# B&R Automation Studio project CControl_Gschneitner (part 4)

#### fbTrockVariante.st - Auswertung der Anlagenkonfiguration mit Ausgabe einer Nummer und eines Textes
```iecst
(********************************************************************
 * COPYRIGHT -- LASCO Heu- und Forsttechnik GmbH
 ********************************************************************
 * Library: LascoTrock
 * Datei: fbTrockVariante.st
 * Autor: Rudolf Lachner
 * Erstellt: 12. Februar 2015
 ********************************************************************
 * Implementierung der Library LascoTrock
 ********************************************************************)

(* Auswertung der Anlagenkonfiguration mit Ausgabe einer Nummer und eines Textes *)
FUNCTION_BLOCK fbTrockVariante

	IF Freigabe THEN

		IF (Ventilator1 AND NOT Ventilator2 AND NOT Luftentfeuchter AND NOT Warmluftofen AND NOT BetriebsmldgWarmluftofen AND NOT BetriebsmldgScheitholzofen AND NOT Brandschutzklappe AND NOT Umschaltklappe) THEN
			VarianteNr 	:= 1;
		ELSIF (Ventilator1 AND NOT Ventilator2 AND NOT Luftentfeuchter AND NOT Warmluftofen AND NOT BetriebsmldgWarmluftofen AND NOT BetriebsmldgScheitholzofen AND NOT Brandschutzklappe AND Umschaltklappe) THEN
			VarianteNr 	:= 2;
		ELSIF (Ventilator1 AND NOT Ventilator2 AND NOT Luftentfeuchter AND NOT Warmluftofen AND NOT BetriebsmldgWarmluftofen AND BetriebsmldgScheitholzofen AND NOT Brandschutzklappe AND NOT Umschaltklappe) THEN
			VarianteNr 	:= 3;
		ELSIF (Ventilator1 AND NOT Ventilator2 AND NOT Luftentfeuchter AND NOT Warmluftofen AND NOT BetriebsmldgWarmluftofen AND BetriebsmldgScheitholzofen AND NOT Brandschutzklappe AND Umschaltklappe) THEN
			VarianteNr 	:= 4;
		ELSIF (Ventilator1 AND NOT Ventilator2 AND NOT Luftentfeuchter AND NOT Warmluftofen AND NOT BetriebsmldgWarmluftofen AND BetriebsmldgScheitholzofen AND Brandschutzklappe AND NOT Umschaltklappe) THEN
			VarianteNr 	:= 5;
		ELSIF (Ventilator1 AND NOT Ventilator2 AND NOT Luftentfeuchter AND NOT Warmluftofen AND NOT BetriebsmldgWarmluftofen AND BetriebsmldgScheitholzofen AND Brandschutzklappe AND Umschaltklappe) THEN
			VarianteNr 	:= 6;
		ELSIF (Ventilator1 AND NOT Ventilator2 AND NOT Luftentfeuchter AND NOT Warmluftofen AND BetriebsmldgWarmluftofen AND NOT BetriebsmldgScheitholzofen AND NOT Brandschutzklappe AND NOT Umschaltklappe) THEN
			VarianteNr 	:= 7;
		ELSIF (Ventilator1 AND NOT Ventilator2 AND NOT Luftentfeuchter AND NOT Warmluftofen AND BetriebsmldgWarmluftofen AND NOT BetriebsmldgScheitholzofen AND NOT Brandschutzklappe AND Umschaltklappe) THEN
			VarianteNr 	:= 8;
		ELSIF (Ventilator1 AND NOT Ventilator2 AND NOT Luftentfeuchter AND NOT Warmluftofen AND BetriebsmldgWarmluftofen AND NOT BetriebsmldgScheitholzofen AND Brandschutzklappe AND NOT Umschaltklappe) THEN
			VarianteNr 	:= 9;
		ELSIF (Ventilator1 AND NOT Ventilator2 AND NOT Luftentfeuchter AND NOT Warmluftofen AND BetriebsmldgWarmluftofen AND NOT BetriebsmldgScheitholzofen AND Brandschutzklappe AND Umschaltklappe) THEN
			VarianteNr 	:= 10;
		ELSIF (Ventilator1 AND NOT Ventilator2 AND NOT Luftentfeuchter AND NOT Warmluftofen AND BetriebsmldgWarmluftofen AND BetriebsmldgScheitholzofen AND NOT Brandschutzklappe AND NOT Umschaltklappe) THEN
			VarianteNr 	:= 11;
		ELSIF (Ventilator1 AND NOT Ventilator2 AND NOT Luftentfeuchter AND NOT Warmluftofen AND BetriebsmldgWarmluftofen AND BetriebsmldgScheitholzofen AND NOT Brandschutzklappe AND Umschaltklappe) THEN
			VarianteNr 	:= 12;
		ELSIF (Ventilator1 AND NOT Ventilator2 AND NOT Luftentfeuchter AND NOT Warmluftofen AND BetriebsmldgWarmluftofen AND BetriebsmldgScheitholzofen AND Brandschutzklappe AND NOT Umschaltklappe) THEN
			VarianteNr 	:= 13;
		ELSIF (Ventilator1 AND NOT Ventilator2 AND NOT Luftentfeuchter AND NOT Warmluftofen AND BetriebsmldgWarmluftofen AND BetriebsmldgScheitholzofen AND Brandschutzklappe AND Umschaltklappe) THEN
			VarianteNr 	:= 14;
		ELSIF (Ventilator1 AND NOT Ventilator2 AND NOT Luftentfeuchter AND Warmluftofen AND NOT BetriebsmldgWarmluftofen AND NOT BetriebsmldgScheitholzofen AND NOT Brandschutzklappe AND NOT Umschaltklappe) THEN
			VarianteNr 	:= 15;
		ELSIF (Ventilator1 AND NOT Ventilator2 AND NOT Luftentfeuchter AND Warmluftofen AND NOT BetriebsmldgWarmluftofen AND NOT BetriebsmldgScheitholzofen AND NOT Brandschutzklappe AND Umschaltklappe) THEN
			VarianteNr 	:= 16;
		ELSIF (Ventilator1 AND NOT Ventilator2 AND NOT Luftentfeuchter AND Warmluftofen AND NOT BetriebsmldgWarmluftofen AND NOT BetriebsmldgScheitholzofen AND Brandschutzklappe AND NOT Umschaltklappe) THEN
			VarianteNr 	:= 17;
		ELSIF (Ventilator1 AND NOT Ventilator2 AND NOT Luftentfeuchter AND Warmluftofen AND NOT BetriebsmldgWarmluftofen AND NOT BetriebsmldgScheitholzofen AND Brandschutzklappe AND Umschaltklappe) THEN
			VarianteNr 	:= 18;
		ELSIF (Ventilator1 AND NOT Ventilator2 AND NOT Luftentfeuchter AND Warmluftofen AND NOT BetriebsmldgWarmluftofen AND BetriebsmldgScheitholzofen AND NOT Brandschutzklappe AND NOT Umschaltklappe) THEN
			VarianteNr 	:= 19;
		ELSIF (Ventilator1 AND NOT Ventilator2 AND NOT Luftentfeuchter AND Warmluftofen AND NOT BetriebsmldgWarmluftofen AND BetriebsmldgScheitholzofen AND NOT Brandschutzklappe AND Umschaltklappe) THEN
			VarianteNr 	:= 20;
		ELSIF (Ventilator1 AND NOT Ventilator2 AND NOT Luftentfeuchter AND Warmluftofen AND NOT BetriebsmldgWarmluftofen AND BetriebsmldgScheitholzofen AND Brandschutzklappe AND NOT Umschaltklappe) THEN
			VarianteNr 	:= 21;
		ELSIF (Ventilator1 AND NOT Ventilator2 AND NOT Luftentfeuchter AND Warmluftofen AND NOT BetriebsmldgWarmluftofen AND BetriebsmldgScheitholzofen AND Brandschutzklappe AND Umschaltklappe) THEN
			VarianteNr 	:= 22;
		ELSIF (Ventilator1 AND NOT Ventilator2 AND NOT Luftentfeuchter AND Warmluftofen AND BetriebsmldgWarmluftofen AND NOT BetriebsmldgScheitholzofen AND NOT Brandschutzklappe AND NOT Umschaltklappe) THEN
			VarianteNr 	:= 23;
		ELSIF (Ventilator1 AND NOT Ventilator2 AND NOT Luftentfeuchter AND Warmluftofen AND BetriebsmldgWarmluftofen AND NOT BetriebsmldgScheitholzofen AND NOT Brandschutzklappe AND Umschaltklappe) THEN
			VarianteNr 	:= 24;
		ELSIF (Ventilator1 AND NOT Ventilator2 AND NOT Luftentfeuchter AND Warmluftofen AND BetriebsmldgWarmluftofen AND NOT BetriebsmldgScheitholzofen AND Brandschutzklappe AND NOT Umschaltklappe) THEN
			VarianteNr 	:= 25;
		ELSIF (Ventilator1 AND NOT Ventilator2 AND NOT Luftentfeuchter AND Warmluftofen AND BetriebsmldgWarmluftofen AND NOT BetriebsmldgScheitholzofen AND Brandschutzklappe AND Umschaltklappe) THEN
			VarianteNr 	:= 26;
		ELSIF (Ventilator1 AND NOT Ventilator2 AND NOT Luftentfeuchter AND Warmluftofen AND BetriebsmldgWarmluftofen AND BetriebsmldgScheitholzofen AND NOT Brandschutzklappe AND NOT Umschaltklappe) THEN
			VarianteNr 	:= 27;
		ELSIF (Ventilator1 AND NOT Ventilator2 AND NOT Luftentfeuchter AND Warmluftofen AND BetriebsmldgWarmluftofen AND BetriebsmldgScheitholzofen AND NOT Brandschutzklappe AND Umschaltklappe) THEN
			VarianteNr 	:= 28;
		ELSIF (Ventilator1 AND NOT Ventilator2 AND NOT Luftentfeuchter AND Warmluftofen AND BetriebsmldgWarmluftofen AND BetriebsmldgScheitholzofen AND Brandschutzklappe AND NOT Umschaltklappe) THEN
			VarianteNr 	:= 29;
		ELSIF (Ventilator1 AND NOT Ventilator2 AND NOT Luftentfeuchter AND Warmluftofen AND BetriebsmldgWarmluftofen AND BetriebsmldgScheitholzofen AND Brandschutzklappe AND Umschaltklappe) THEN
			VarianteNr 	:= 30;
		ELSIF (Ventilator1 AND NOT Ventilator2 AND Luftentfeuchter AND NOT Warmluftofen AND NOT BetriebsmldgWarmluftofen AND NOT BetriebsmldgScheitholzofen AND NOT Brandschutzklappe AND NOT Umschaltklappe) THEN
			VarianteNr 	:= 31;
		ELSIF (Ventilator1 AND NOT Ventilator2 AND Luftentfeuchter AND NOT Warmluftofen AND NOT BetriebsmldgWarmluftofen AND NOT BetriebsmldgScheitholzofen AND NOT Brandschutzklappe AND Umschaltklappe) THEN
			VarianteNr 	:= 32;
		ELSIF (Ventilator1 AND NOT Ventilator2 AND Luftentfeuchter AND NOT Warmluftofen AND NOT BetriebsmldgWarmluftofen AND BetriebsmldgScheitholzofen AND NOT Brandschutzklappe AND NOT Umschaltklappe) THEN
			VarianteNr 	:= 33;
		ELSIF (Ventilator1 AND NOT Ventilator2 AND Luftentfeuchter AND NOT Warmluftofen AND NOT BetriebsmldgWarmluftofen AND BetriebsmldgScheitholzofen AND NOT Brandschutzklappe AND Umschaltklappe) THEN
			VarianteNr 	:= 34;
		ELSIF (Ventilator1 AND NOT Ventilator2 AND Luftentfeuchter AND NOT Warmluftofen AND NOT BetriebsmldgWarmluftofen AND BetriebsmldgScheitholzofen AND Brandschutzklappe AND NOT Umschaltklappe) THEN
			VarianteNr 	:= 35;
		ELSIF (Ventilator1 AND NOT Ventilator2 AND Luftentfeuchter AND NOT Warmluftofen AND NOT BetriebsmldgWarmluftofen AND BetriebsmldgScheitholzofen AND Brandschutzklappe AND Umschaltklappe) THEN
			VarianteNr 	:= 36;
		ELSIF (Ventilator1 AND NOT Ventilator2 AND Luftentfeuchter AND NOT Warmluftofen AND BetriebsmldgWarmluftofen AND NOT BetriebsmldgScheitholzofen AND NOT Brandschutzklappe AND NOT Umschaltklappe) THEN
			VarianteNr 	:= 37;
		ELSIF (Ventilator1 AND NOT Ventilator2 AND Luftentfeuchter AND NOT Warmluftofen AND BetriebsmldgWarmluftofen AND NOT BetriebsmldgScheitholzofen AND NOT Brandschutzklappe AND Umschaltklappe) THEN
			VarianteNr 	:= 38;
		ELSIF (Ventilator1 AND NOT Ventilator2 AND Luftentfeuchter AND NOT Warmluftofen AND BetriebsmldgWarmluftofen AND NOT BetriebsmldgScheitholzofen AND Brandschutzklappe AND NOT Umschaltklappe) THEN
			VarianteNr 	:= 39;
		ELSIF (Ventilator1 AND NOT Ventilator2 AND Luftentfeuchter AND NOT Warmluftofen AND BetriebsmldgWarmluftofen AND NOT BetriebsmldgScheitholzofen AND Brandschutzklappe AND Umschaltklappe) THEN
			VarianteNr 	:= 40;
		ELSIF (Ventilator1 AND NOT Ventilator2 AND Luftentfeuchter AND NOT Warmluftofen AND BetriebsmldgWarmluftofen AND BetriebsmldgScheitholzofen AND NOT Brandschutzklappe AND NOT Umschaltklappe) THEN
			VarianteNr 	:= 41;
		ELSIF (Ventilator1 AND NOT Ventilator2 AND Luftentfeuchter AND NOT Warmluftofen AND BetriebsmldgWarmluftofen AND BetriebsmldgScheitholzofen AND NOT Brandschutzklappe AND Umschaltklappe) THEN
			VarianteNr 	:= 42;
		ELSIF (Ventilator1 AND NOT Ventilator2 AND Luftentfeuchter AND NOT Warmluftofen AND BetriebsmldgWarmluftofen AND BetriebsmldgScheitholzofen AND Brandschutzklappe AND NOT Umschaltklappe) THEN
			VarianteNr 	:= 43;
		ELSIF (Ventilator1 AND NOT Ventilator2 AND Luftentfeuchter AND NOT Warmluftofen AND BetriebsmldgWarmluftofen AND BetriebsmldgScheitholzofen AND Brandschutzklappe AND Umschaltklappe) THEN
			VarianteNr 	:= 44;
		ELSIF (Ventilator1 AND NOT Ventilator2 AND Luftentfeuchter AND Warmluftofen AND NOT BetriebsmldgWarmluftofen AND NOT BetriebsmldgScheitholzofen AND NOT Brandschutzklappe AND NOT Umschaltklappe) THEN
			VarianteNr 	:= 45;
		ELSIF (Ventilator1 AND NOT Ventilator2 AND Luftentfeuchter AND Warmluftofen AND NOT BetriebsmldgWarmluftofen AND NOT BetriebsmldgScheitholzofen AND NOT Brandschutzklappe AND Umschaltklappe) THEN
			VarianteNr 	:= 46;
		ELSIF (Ventilator1 AND NOT Ventilator2 AND Luftentfeuchter AND Warmluftofen AND NOT BetriebsmldgWarmluftofen AND NOT BetriebsmldgScheitholzofen AND Brandschutzklappe AND NOT Umschaltklappe) THEN
			VarianteNr 	:= 47;
		ELSIF (Ventilator1 AND NOT Ventilator2 AND Luftentfeuchter AND Warmluftofen AND NOT BetriebsmldgWarmluftofen AND NOT BetriebsmldgScheitholzofen AND Brandschutzklappe AND Umschaltklappe) THEN
			VarianteNr 	:= 48;
		ELSIF (Ventilator1 AND NOT Ventilator2 AND Luftentfeuchter AND Warmluftofen AND NOT BetriebsmldgWarmluftofen AND BetriebsmldgScheitholzofen AND NOT Brandschutzklappe AND NOT Umschaltklappe) THEN
			VarianteNr 	:= 49;
		ELSIF (Ventilator1 AND NOT Ventilator2 AND Luftentfeuchter AND Warmluftofen AND NOT BetriebsmldgWarmluftofen AND BetriebsmldgScheitholzofen AND NOT Brandschutzklappe AND Umschaltklappe) THEN
			VarianteNr 	:= 50;
		ELSIF (Ventilator1 AND NOT Ventilator2 AND Luftentfeuchter AND Warmluftofen AND NOT BetriebsmldgWarmluftofen AND BetriebsmldgScheitholzofen AND Brandschutzklappe AND NOT Umschaltklappe) THEN
			VarianteNr 	:= 51;
		ELSIF (Ventilator1 AND NOT Ventilator2 AND Luftentfeuchter AND Warmluftofen AND NOT BetriebsmldgWarmluftofen AND BetriebsmldgScheitholzofen AND Brandschutzklappe AND Umschaltklappe) THEN
			VarianteNr 	:= 52;
		ELSIF (Ventilator1 AND NOT Ventilator2 AND Luftentfeuchter AND Warmluftofen AND BetriebsmldgWarmluftofen AND NOT BetriebsmldgScheitholzofen AND NOT Brandschutzklappe AND NOT Umschaltklappe) THEN
			VarianteNr 	:= 53;
		ELSIF (Ventilator1 AND NOT Ventilator2 AND Luftentfeuchter AND Warmluftofen AND BetriebsmldgWarmluftofen AND NOT BetriebsmldgScheitholzofen AND NOT Brandschutzklappe AND Umschaltklappe) THEN
			VarianteNr 	:= 54;
		ELSIF (Ventilator1 AND NOT Ventilator2 AND Luftentfeuchter AND Warmluftofen AND BetriebsmldgWarmluftofen AND NOT BetriebsmldgScheitholzofen AND Brandschutzklappe AND NOT Umschaltklappe) THEN
			VarianteNr 	:= 55;
		ELSIF (Ventilator1 AND NOT Ventilator2 AND Luftentfeuchter AND Warmluftofen AND BetriebsmldgWarmluftofen AND NOT BetriebsmldgScheitholzofen AND Brandschutzklappe AND Umschaltklappe) THEN
			VarianteNr 	:= 56;
		ELSIF (Ventilator1 AND NOT Ventilator2 AND Luftentfeuchter AND Warmluftofen AND BetriebsmldgWarmluftofen AND BetriebsmldgScheitholzofen AND NOT Brandschutzklappe AND NOT Umschaltklappe) THEN
			VarianteNr 	:= 57;
		ELSIF (Ventilator1 AND NOT Ventilator2 AND Luftentfeuchter AND Warmluftofen AND BetriebsmldgWarmluftofen AND BetriebsmldgScheitholzofen AND NOT Brandschutzklappe AND Umschaltklappe) THEN
			VarianteNr 	:= 58;
		ELSIF (Ventilator1 AND NOT Ventilator2 AND Luftentfeuchter AND Warmluftofen AND BetriebsmldgWarmluftofen AND BetriebsmldgScheitholzofen AND Brandschutzklappe AND NOT Umschaltklappe) THEN
			VarianteNr 	:= 59;
		ELSIF (Ventilator1 AND NOT Ventilator2 AND Luftentfeuchter AND Warmluftofen AND BetriebsmldgWarmluftofen AND BetriebsmldgScheitholzofen AND Brandschutzklappe AND Umschaltklappe) THEN
			VarianteNr 	:= 60;
		ELSIF (Ventilator1 AND Ventilator2 AND NOT Luftentfeuchter AND NOT Warmluftofen AND NOT BetriebsmldgWarmluftofen AND NOT BetriebsmldgScheitholzofen AND NOT Brandschutzklappe AND NOT Umschaltklappe) THEN
			VarianteNr 	:= 61;
		ELSIF (Ventilator1 AND Ventilator2 AND NOT Luftentfeuchter AND NOT Warmluftofen AND NOT BetriebsmldgWarmluftofen AND NOT BetriebsmldgScheitholzofen AND NOT Brandschutzklappe AND Umschaltklappe) THEN
			VarianteNr 	:= 62;
		ELSIF (Ventilator1 AND Ventilator2 AND NOT Luftentfeuchter AND NOT Warmluftofen AND NOT BetriebsmldgWarmluftofen AND BetriebsmldgScheitholzofen AND NOT Brandschutzklappe AND NOT Umschaltklappe) THEN
			VarianteNr 	:= 63;
		ELSIF (Ventilator1 AND Ventilator2 AND NOT Luftentfeuchter AND NOT Warmluftofen AND NOT BetriebsmldgWarmluftofen AND BetriebsmldgScheitholzofen AND NOT Brandschutzklappe AND Umschaltklappe) THEN
			VarianteNr 	:= 64;
		ELSIF (Ventilator1 AND Ventilator2 AND NOT Luftentfeuchter AND NOT Warmluftofen AND NOT BetriebsmldgWarmluftofen AND BetriebsmldgScheitholzofen AND Brandschutzklappe AND NOT Umschaltklappe) THEN
			VarianteNr 	:= 65;
		ELSIF (Ventilator1 AND Ventilator2 AND NOT Luftentfeuchter AND NOT Warmluftofen AND NOT BetriebsmldgWarmluftofen AND BetriebsmldgScheitholzofen AND Brandschutzklappe AND Umschaltklappe) THEN
			VarianteNr 	:= 66;
		ELSIF (Ventilator1 AND Ventilator2 AND NOT Luftentfeuchter AND NOT Warmluftofen AND BetriebsmldgWarmluftofen AND NOT BetriebsmldgScheitholzofen AND NOT Brandschutzklappe AND NOT Umschaltklappe) THEN
			VarianteNr 	:= 67;
		ELSIF (Ventilator1 AND Ventilator2 AND NOT Luftentfeuchter AND NOT Warmluftofen AND BetriebsmldgWarmluftofen AND NOT BetriebsmldgScheitholzofen AND NOT Brandschutzklappe AND Umschaltklappe) THEN
			VarianteNr 	:= 68;
		ELSIF (Ventilator1 AND Ventilator2 AND NOT Luftentfeuchter AND NOT Warmluftofen AND BetriebsmldgWarmluftofen AND NOT BetriebsmldgScheitholzofen AND Brandschutzklappe AND NOT Umschaltklappe) THEN
			VarianteNr 	:= 69;
		ELSIF (Ventilator1 AND Ventilator2 AND NOT Luftentfeuchter AND NOT Warmluftofen AND BetriebsmldgWarmluftofen AND NOT BetriebsmldgScheitholzofen AND Brandschutzklappe AND Umschaltklappe) THEN
			VarianteNr 	:= 70;
		ELSIF (Ventilator1 AND Ventilator2 AND NOT Luftentfeuchter AND NOT Warmluftofen AND BetriebsmldgWarmluftofen AND BetriebsmldgScheitholzofen AND NOT Brandschutzklappe AND NOT Umschaltklappe) THEN
			VarianteNr 	:= 71;
		ELSIF (Ventilator1 AND Ventilator2 AND NOT Luftentfeuchter AND NOT Warmluftofen AND BetriebsmldgWarmluftofen AND BetriebsmldgScheitholzofen AND NOT Brandschutzklappe AND Umschaltklappe) THEN
			VarianteNr 	:= 72;
		ELSIF (Ventilator1 AND Ventilator2 AND NOT Luftentfeuchter AND NOT Warmluftofen AND BetriebsmldgWarmluftofen AND BetriebsmldgScheitholzofen AND Brandschutzklappe AND NOT Umschaltklappe) THEN
			VarianteNr 	:= 73;
		ELSIF (Ventilator1 AND Ventilator2 AND NOT Luftentfeuchter AND NOT Warmluftofen AND BetriebsmldgWarmluftofen AND BetriebsmldgScheitholzofen AND Brandschutzklappe AND Umschaltklappe) THEN
			VarianteNr 	:= 74;
		ELSIF (Ventilator1 AND Ventilator2 AND NOT Luftentfeuchter AND Warmluftofen AND NOT BetriebsmldgWarmluftofen AND NOT BetriebsmldgScheitholzofen AND NOT Brandschutzklappe AND NOT Umschaltklappe) THEN
			VarianteNr 	:= 75;
		ELSIF (Ventilator1 AND Ventilator2 AND NOT Luftentfeuchter AND Warmluftofen AND NOT BetriebsmldgWarmluftofen AND NOT BetriebsmldgScheitholzofen AND NOT Brandschutzklappe AND Umschaltklappe) THEN
			VarianteNr 	:= 76;
		ELSIF (Ventilator1 AND Ventilator2 AND NOT Luftentfeuchter AND Warmluftofen AND NOT BetriebsmldgWarmluftofen AND NOT BetriebsmldgScheitholzofen AND Brandschutzklappe AND NOT Umschaltklappe) THEN
			VarianteNr 	:= 77;
		ELSIF (Ventilator1 AND Ventilator2 AND NOT Luftentfeuchter AND Warmluftofen AND NOT BetriebsmldgWarmluftofen AND NOT BetriebsmldgScheitholzofen AND Brandschutzklappe AND Umschaltklappe) THEN
			VarianteNr 	:= 78;
		ELSIF (Ventilator1 AND Ventilator2 AND NOT Luftentfeuchter AND Warmluftofen AND NOT BetriebsmldgWarmluftofen AND BetriebsmldgScheitholzofen AND NOT Brandschutzklappe AND NOT Umschaltklappe) THEN
			VarianteNr 	:= 79;
		ELSIF (Ventilator1 AND Ventilator2 AND NOT Luftentfeuchter AND Warmluftofen AND NOT BetriebsmldgWarmluftofen AND BetriebsmldgScheitholzofen AND NOT Brandschutzklappe AND Umschaltklappe) THEN
			VarianteNr 	:= 80;
		ELSIF (Ventilator1 AND Ventilator2 AND NOT Luftentfeuchter AND Warmluftofen AND NOT BetriebsmldgWarmluftofen AND BetriebsmldgScheitholzofen AND Brandschutzklappe AND NOT Umschaltklappe) THEN
			VarianteNr 	:= 81;
		ELSIF (Ventilator1 AND Ventilator2 AND NOT Luftentfeuchter AND Warmluftofen AND NOT BetriebsmldgWarmluftofen AND BetriebsmldgScheitholzofen AND Brandschutzklappe AND Umschaltklappe) THEN
			VarianteNr 	:= 82;
		ELSIF (Ventilator1 AND Ventilator2 AND NOT Luftentfeuchter AND Warmluftofen AND BetriebsmldgWarmluftofen AND NOT BetriebsmldgScheitholzofen AND NOT Brandschutzklappe AND NOT Umschaltklappe) THEN
			VarianteNr 	:= 83;
		ELSIF (Ventilator1 AND Ventilator2 AND NOT Luftentfeuchter AND Warmluftofen AND BetriebsmldgWarmluftofen AND NOT BetriebsmldgScheitholzofen AND NOT Brandschutzklappe AND Umschaltklappe) THEN
			VarianteNr 	:= 84;
		ELSIF (Ventilator1 AND Ventilator2 AND NOT Luftentfeuchter AND Warmluftofen AND BetriebsmldgWarmluftofen AND NOT BetriebsmldgScheitholzofen AND Brandschutzklappe AND NOT Umschaltklappe) THEN
			VarianteNr 	:= 85;
		ELSIF (Ventilator1 AND Ventilator2 AND NOT Luftentfeuchter AND Warmluftofen AND BetriebsmldgWarmluftofen AND NOT BetriebsmldgScheitholzofen AND Brandschutzklappe AND Umschaltklappe) THEN
			VarianteNr 	:= 86;
		ELSIF (Ventilator1 AND Ventilator2 AND NOT Luftentfeuchter AND Warmluftofen AND BetriebsmldgWarmluftofen AND BetriebsmldgScheitholzofen AND NOT Brandschutzklappe AND NOT Umschaltklappe) THEN
			VarianteNr 	:= 87;
		ELSIF (Ventilator1 AND Ventilator2 AND NOT Luftentfeuchter AND Warmluftofen AND BetriebsmldgWarmluftofen AND BetriebsmldgScheitholzofen AND NOT Brandschutzklappe AND Umschaltklappe) THEN
			VarianteNr 	:= 88;
		ELSIF (Ventilator1 AND Ventilator2 AND NOT Luftentfeuchter AND Warmluftofen AND BetriebsmldgWarmluftofen AND BetriebsmldgScheitholzofen AND Brandschutzklappe AND NOT Umschaltklappe) THEN
			VarianteNr 	:= 89;
		ELSIF (Ventilator1 AND Ventilator2 AND NOT Luftentfeuchter AND Warmluftofen AND BetriebsmldgWarmluftofen AND BetriebsmldgScheitholzofen AND Brandschutzklappe AND Umschaltklappe) THEN
			VarianteNr 	:= 90;
		ELSIF (Ventilator1 AND Ventilator2 AND Luftentfeuchter AND NOT Warmluftofen AND NOT BetriebsmldgWarmluftofen AND NOT BetriebsmldgScheitholzofen AND NOT Brandschutzklappe AND NOT Umschaltklappe) THEN
			VarianteNr 	:= 91;
		ELSIF (Ventilator1 AND Ventilator2 AND Luftentfeuchter AND NOT Warmluftofen AND NOT BetriebsmldgWarmluftofen AND NOT BetriebsmldgScheitholzofen AND NOT Brandschutzklappe AND Umschaltklappe) THEN
			VarianteNr 	:= 92;
		ELSIF (Ventilator1 AND Ventilator2 AND Luftentfeuchter AND NOT Warmluftofen AND NOT BetriebsmldgWarmluftofen AND BetriebsmldgScheitholzofen AND NOT Brandschutzklappe AND NOT Umschaltklappe) THEN
			VarianteNr 	:= 93;
		ELSIF (Ventilator1 AND Ventilator2 AND Luftentfeuchter AND NOT Warmluftofen AND NOT BetriebsmldgWarmluftofen AND BetriebsmldgScheitholzofen AND NOT Brandschutzklappe AND Umschaltklappe) THEN
			VarianteNr 	:= 94;
		ELSIF (Ventilator1 AND Ventilator2 AND Luftentfeuchter AND NOT Warmluftofen AND NOT BetriebsmldgWarmluftofen AND BetriebsmldgScheitholzofen AND Brandschutzklappe AND NOT Umschaltklappe) THEN
			VarianteNr 	:= 95;
		ELSIF (Ventilator1 AND Ventilator2 AND Luftentfeuchter AND NOT Warmluftofen AND NOT BetriebsmldgWarmluftofen AND BetriebsmldgScheitholzofen AND Brandschutzklappe AND Umschaltklappe) THEN
			VarianteNr 	:= 96;
		ELSIF (Ventilator1 AND Ventilator2 AND Luftentfeuchter AND NOT Warmluftofen AND BetriebsmldgWarmluftofen AND NOT BetriebsmldgScheitholzofen AND NOT Brandschutzklappe AND NOT Umschaltklappe) THEN
			VarianteNr 	:= 97;
		ELSIF (Ventilator1 AND Ventilator2 AND Luftentfeuchter AND NOT Warmluftofen AND BetriebsmldgWarmluftofen AND NOT BetriebsmldgScheitholzofen AND NOT Brandschutzklappe AND Umschaltklappe) THEN
			VarianteNr 	:= 98;
		ELSIF (Ventilator1 AND Ventilator2 AND Luftentfeuchter AND NOT Warmluftofen AND BetriebsmldgWarmluftofen AND NOT BetriebsmldgScheitholzofen AND Brandschutzklappe AND NOT Umschaltklappe) THEN
			VarianteNr 	:= 99;
		ELSIF (Ventilator1 AND Ventilator2 AND Luftentfeuchter AND NOT Warmluftofen AND BetriebsmldgWarmluftofen AND NOT BetriebsmldgScheitholzofen AND Brandschutzklappe AND Umschaltklappe) THEN
			VarianteNr 	:= 100;
		ELSIF (Ventilator1 AND Ventilator2 AND Luftentfeuchter AND NOT Warmluftofen AND BetriebsmldgWarmluftofen AND BetriebsmldgScheitholzofen AND NOT Brandschutzklappe AND NOT Umschaltklappe) THEN
			VarianteNr 	:= 101;
		ELSIF (Ventilator1 AND Ventilator2 AND Luftentfeuchter AND NOT Warmluftofen AND BetriebsmldgWarmluftofen AND BetriebsmldgScheitholzofen AND NOT Brandschutzklappe AND Umschaltklappe) THEN
			VarianteNr 	:= 102;
		ELSIF (Ventilator1 AND Ventilator2 AND Luftentfeuchter AND NOT Warmluftofen AND BetriebsmldgWarmluftofen AND BetriebsmldgScheitholzofen AND Brandschutzklappe AND NOT Umschaltklappe) THEN
			VarianteNr 	:= 103;
		ELSIF (Ventilator1 AND Ventilator2 AND Luftentfeuchter AND NOT Warmluftofen AND BetriebsmldgWarmluftofen AND BetriebsmldgScheitholzofen AND Brandschutzklappe AND Umschaltklappe) THEN
			VarianteNr 	:= 104;
		ELSIF (Ventilator1 AND Ventilator2 AND Luftentfeuchter AND Warmluftofen AND NOT BetriebsmldgWarmluftofen AND NOT BetriebsmldgScheitholzofen AND NOT Brandschutzklappe AND NOT Umschaltklappe) THEN
			VarianteNr 	:= 105;
		ELSIF (Ventilator1 AND Ventilator2 AND Luftentfeuchter AND Warmluftofen AND NOT BetriebsmldgWarmluftofen AND NOT BetriebsmldgScheitholzofen AND NOT Brandschutzklappe AND Umschaltklappe) THEN
			VarianteNr 	:= 106;
		ELSIF (Ventilator1 AND Ventilator2 AND Luftentfeuchter AND Warmluftofen AND NOT BetriebsmldgWarmluftofen AND NOT BetriebsmldgScheitholzofen AND Brandschutzklappe AND NOT Umschaltklappe) THEN
			VarianteNr 	:= 107;
		ELSIF (Ventilator1 AND Ventilator2 AND Luftentfeuchter AND Warmluftofen AND NOT BetriebsmldgWarmluftofen AND NOT BetriebsmldgScheitholzofen AND Brandschutzklappe AND Umschaltklappe) THEN
			VarianteNr 	:= 108;
		ELSIF (Ventilator1 AND Ventilator2 AND Luftentfeuchter AND Warmluftofen AND NOT BetriebsmldgWarmluftofen AND BetriebsmldgScheitholzofen AND NOT Brandschutzklappe AND NOT Umschaltklappe) THEN
			VarianteNr 	:= 109;
		ELSIF (Ventilator1 AND Ventilator2 AND Luftentfeuchter AND Warmluftofen AND NOT BetriebsmldgWarmluftofen AND BetriebsmldgScheitholzofen AND NOT Brandschutzklappe AND Umschaltklappe) THEN
			VarianteNr 	:= 110;
		ELSIF (Ventilator1 AND Ventilator2 AND Luftentfeuchter AND Warmluftofen AND NOT BetriebsmldgWarmluftofen AND BetriebsmldgScheitholzofen AND Brandschutzklappe AND NOT Umschaltklappe) THEN
			VarianteNr 	:= 111;
		ELSIF (Ventilator1 AND Ventilator2 AND Luftentfeuchter AND Warmluftofen AND NOT BetriebsmldgWarmluftofen AND BetriebsmldgScheitholzofen AND Brandschutzklappe AND Umschaltklappe) THEN
			VarianteNr 	:= 112;
		ELSIF (Ventilator1 AND Ventilator2 AND Luftentfeuchter AND Warmluftofen AND BetriebsmldgWarmluftofen AND NOT BetriebsmldgScheitholzofen AND NOT Brandschutzklappe AND NOT Umschaltklappe) THEN
			VarianteNr 	:= 113;
		ELSIF (Ventilator1 AND Ventilator2 AND Luftentfeuchter AND Warmluftofen AND BetriebsmldgWarmluftofen AND NOT BetriebsmldgScheitholzofen AND NOT Brandschutzklappe AND Umschaltklappe) THEN
			VarianteNr 	:= 114;
		ELSIF (Ventilator1 AND Ventilator2 AND Luftentfeuchter AND Warmluftofen AND BetriebsmldgWarmluftofen AND NOT BetriebsmldgScheitholzofen AND Brandschutzklappe AND NOT Umschaltklappe) THEN
			VarianteNr 	:= 115;
		ELSIF (Ventilator1 AND Ventilator2 AND Luftentfeuchter AND Warmluftofen AND BetriebsmldgWarmluftofen AND NOT BetriebsmldgScheitholzofen AND Brandschutzklappe AND Umschaltklappe) THEN
			VarianteNr 	:= 116;
		ELSIF (Ventilator1 AND Ventilator2 AND Luftentfeuchter AND Warmluftofen AND BetriebsmldgWarmluftofen AND BetriebsmldgScheitholzofen AND NOT Brandschutzklappe AND NOT Umschaltklappe) THEN
			VarianteNr 	:= 117;
		ELSIF (Ventilator1 AND Ventilator2 AND Luftentfeuchter AND Warmluftofen AND BetriebsmldgWarmluftofen AND BetriebsmldgScheitholzofen AND NOT Brandschutzklappe AND Umschaltklappe) THEN
			VarianteNr 	:= 118;
		ELSIF (Ventilator1 AND Ventilator2 AND Luftentfeuchter AND Warmluftofen AND BetriebsmldgWarmluftofen AND BetriebsmldgScheitholzofen AND Brandschutzklappe AND NOT Umschaltklappe) THEN
			VarianteNr 	:= 119;
		ELSIF (Ventilator1 AND Ventilator2 AND Luftentfeuchter AND Warmluftofen AND BetriebsmldgWarmluftofen AND BetriebsmldgScheitholzofen AND Brandschutzklappe AND Umschaltklappe) THEN
			VarianteNr 	:= 120;
		ELSE
			VarianteNr	:= 0;
		END_IF

	//	VarianteName	:= TROCK_VARIANTEN_NAMEN[VarianteNr];

	ELSE

		VarianteNr		:= 0;
	//	VarianteName	:= TROCK_VARIANTEN_NAMEN[VarianteNr];

	END_IF

END_FUNCTION_BLOCK
```

### Library Logical/Libraries/LascoUtil (IEC, version 1.00.0) - Eine neue Quellbibliothek
Depends on: LoopConR

#### LascoUtil.typ - Exportierte Datentypen
```iecst
(********************************************************************
 * COPYRIGHT -- LASCO Heu- und Forsttechnik GmbH
 ********************************************************************
 * Library: LascoUtil
 * Datei: LascoUtil.typ
 * Autor: Rudolf Lachner
 * Erstellt: 27. März 2013
 ********************************************************************
 * Datentypen der Library LascoUtil
 ********************************************************************)

TYPE
	WoPrg_type : 	STRUCT
		HZ1_Enable : BOOL;
		HZ2_Enable : BOOL;
		HZ1_Std_Ein : REAL;
		HZ1_Min_Ein : REAL;
		HZ1_Std_Aus : REAL;
		HZ1_Min_Aus : REAL;
		HZ2_Std_Ein : REAL;
		HZ2_Min_Ein : REAL;
		HZ2_Std_Aus : REAL;
		HZ2_Min_Aus : REAL;
	END_STRUCT;
	Zeit_type : 	STRUCT
		Jahr : UINT;
		Monat : USINT;
		Tag : USINT;
		WoTag : USINT;
		Stunde : USINT;
		Minute : USINT;
		Sekunde : USINT;
		Milli : UINT;
		Mikro : UINT;
	END_STRUCT;
	enumStepsBskUeberw :
		(
		BSK_WARTEN := 0,
		BSK_OEFFNEN := 1,
		BSK_OEFFNEN_FEHLER := 2,
		BSK_SCHLIESSEN := 3,
		BSK_SCHLIESSEN_FEHLER := 4,
		BSK_STOERUNG := 5
		);
END_TYPE
```

#### LascoUtil.fun - Exportierte Funktionen und Funktionsblöcke
```iecst
(********************************************************************
 * COPYRIGHT -- LASCO Heu- und Forsttechnik GmbH
 ********************************************************************
 * Library: LascoUtil
 * Datei: LascoUtil.fun
 * Autor: Rudolf Lachner
 * Erstellt: 27. März 2013
 ********************************************************************
 * Funktionen und Funktionsblöcke der Library LascoUtil
 ********************************************************************)

FUNCTION_BLOCK fbLascoAutoRuecklauf (*Automatische Rücklauffunktion für Motoren*) (*$GROUP=Anwender*)
	VAR_INPUT
		Freigabe : BOOL; (*Freigabe der Funktion*)
		ImpulseVorBisRueck : UDINT; (*Nach dieser Anzahl von Vorwärtsimpulsen fährt der Motor für die Dauer "Rücklaufzeit" zurück.*)
		Ruecklaufzeit : UDINT; (*Rücklaufzeit*)
		VerzUmschaltung : UDINT; (*Verzögerungszeit zwischen Vor und Zurück*)
		ImpulsVor : BOOL; (*Vorwärtsimpuls des Motors*)
		Zuendphase : BOOL; (*Modus Zündphase (1. Einschub)*)
		Heizphase : BOOL; (*Modus Heizphase*)
		LaufzeitEinschubZuendung : UDINT; (*Laufzeit 1. Einschub bei Zündung*)
		sekTick : BOOL; (*Sekundentakt*)
		MaxLaufzeitVor : REAL; (*Max. Laufzeit Vorwärts bei 1. Einschub (danach fährt Schnecke zurück)*)
	END_VAR
	VAR_OUTPUT
		MotorRueck : BOOL; (*Kommando Motor Rückwärts*)
		MotorVor : BOOL;
	END_VAR
	VAR
		ctEinschuebeSeitRuecklauf : UDINT;
		loc_RuecklaufErforderlich : BOOL;
		TON_Umschaltverz : TON;
		zzEdge00000 : BOOL;
		zzEdge00001 : BOOL;
		zzEdge00002 : BOOL;
		TOF_Ruecklauf : TOF;
		loc_curStep : USINT;
		stateEntry : BOOL;
		ctLaufzeitEinschub1 : UDINT;
		ctLaufzeitEinschubVor : UDINT;
		loc_RueckwaertsOk : BOOL;
		zzEdge00003 : BOOL;
		zzEdge00004 : BOOL;
		zzEdge00005 : BOOL;
		zzEdge00006 : BOOL;
	END_VAR
END_FUNCTION_BLOCK

FUNCTION_BLOCK fbLascoBskUeberw (*Ansteuerung Brandschutzklappe mit Laufzeitüberwachung und Freiräumung*) (*$GROUP=Anwender*)
	VAR_INPUT
		Freigabe : BOOL; (*Freigabe Funktionsbaustein*)
		FreigabeOeffnen : BOOL; (*Befehl Klappe Öffnen*)
		FreigabeSchliessen : BOOL; (*Befehl Klappe Schließen*)
		diKlappeGeschlossen : BOOL; (*Eingang Klappe ist geschlossen*)
		diKlappeGeoeffnet : BOOL; (*Eingang Klappe ist geöffnet*)
		Quit : BOOL; (*Fehlerquittierung*)
		MaxVersucheZu : UDINT; (*Max. Versuche Klappe schließen bis Fehlerausgabe*)
		MaxVersucheAuf : UDINT; (*Max. Versuche Klappe öffnen bis Fehlerausgabe*)
		LaufzeitZu : UDINT; (*Laufzeit Klappe schließen [ms]*)
		LaufzeitAuf : UDINT; (*Laufzeit Klappe öffnen [ms]*)
	END_VAR
	VAR_OUTPUT
		doKlappeOeffnen : BOOL; (*Ausgang Klappe öffnen*)
		Stoerung : BOOL; (*Ausgang Störung*)
		ctVersucheAuf : UDINT; (*Zähler Anzahl Fehlversuche Öffnen*)
		ctVersucheZu : UDINT; (*Zähler Anzahl Fehlversuche Schließen*)
	END_VAR
	VAR
		TON_Laufzeit : TON; (*TON Laufzeitüberwachung*)
		stateEntry : BOOL;
		lastStep : enumStepsBskUeberw;
		nextStep : enumStepsBskUeberw;
		curStep : enumStepsBskUeberw;
		loc_KlappeIstOffen : BOOL;
		loc_KlappeIstGeschlossen : BOOL;
	END_VAR
END_FUNCTION_BLOCK

FUNCTION_BLOCK fbLascoEUhr (*Echtzeituhr auslesen*)
	VAR_INPUT
		Freigabe : BOOL;
	END_VAR
	VAR_OUTPUT
		StdMin : INT;
		Jahr : UINT;
		Monat : USINT;
		Tag : USINT;
		WoTag : USINT;
		Stunde : USINT;
		Minute : USINT;
		Sekunde : USINT;
		Milli : UINT;
		Mikro : UINT;
	END_VAR
	VAR
		Echtzeit : Zeit_type;
		DTGetTime_0 : DTGetTime;
		DateTime : DATE_AND_TIME;
	END_VAR
END_FUNCTION_BLOCK

FUNCTION_BLOCK fbLascoTON (*Einschaltverzögerung*)
	VAR_INPUT
		IN : BOOL;
		Zeit : REAL;
		Tick : BOOL;
	END_VAR
	VAR_OUTPUT
		Q : BOOL;
	END_VAR
	VAR
		Elapsed : REAL;
	END_VAR
END_FUNCTION_BLOCK

FUNCTION_BLOCK fbLascoTOF (*Ausschaltverzögerung*)
	VAR_INPUT
		IN : BOOL; (*Freigabe*)
		Reset : BOOL; (*Reset Ausschaltverzögerung*)
		Zeit : REAL; (*Verzögerungszeit*)
		Tick : BOOL; (*Taktfrequeunz*)
	END_VAR
	VAR_OUTPUT
		Q : BOOL; (*Ausgang*)
	END_VAR
	VAR
		Elapsed : REAL;
	END_VAR
END_FUNCTION_BLOCK

FUNCTION_BLOCK fbLascoTOG (*Toggle- Funktion*)
	VAR_INPUT
		IN : BOOL;
		Reset : BOOL;
	END_VAR
	VAR_OUTPUT
		Q : BOOL;
	END_VAR
	VAR
		ToggImp : BOOL;
	END_VAR
END_FUNCTION_BLOCK

FUNCTION funLascoMinss : REAL (*Wert in Minuten und Sekunden umwandeln*)
	VAR_INPUT
		IN : REAL;
	END_VAR
END_FUNCTION

FUNCTION_BLOCK fbLascoZdxx (*Tickausgabe bei Zustandsänderung des Einganges*)
	VAR_INPUT
		IN : REAL; (*Eingangsvariable, die auf eine Veränderung kontrolliert wird*)
	END_VAR
	VAR_OUTPUT
		Q : BOOL; (*Flanke, wenn Änderung am Eingang*)
	END_VAR
	VAR
		MEM : REAL;
	END_VAR
END_FUNCTION_BLOCK

FUNCTION_BLOCK fbLascoZbFrg (*Zeitfenster Freigabe*)
	VAR_INPUT
		Freigabe : BOOL; (*Freigabe*)
		StartZeit : REAL; (*Start-Zeit im Format hhmm*)
		StoppZeit : REAL; (*Stopp-Zeit im Format hhmm*)
	END_VAR
	VAR_OUTPUT
		FreigZeitfenster : BOOL; (*Ausgang Freigabe*)
	END_VAR
	VAR
		EUhr : fbLascoEUhr;
		AktZeit : REAL;
	END_VAR
END_FUNCTION_BLOCK

FUNCTION_BLOCK fbLascoBstd (*Betriebsstundenzähler auf Minutenbasis*)
	VAR_INPUT
		Aktiv : BOOL; (*Betriebsmittel ist Aktiv*)
		minTick : BOOL; (*Minutentakt*)
		Stunden : REFERENCE TO UDINT; (*Betriebsstunden*)
		Reset : BOOL; (*Alles Rücksetzen*)
	END_VAR
	VAR
		Minuten : USINT; (*Minutenzähler*)
	END_VAR
END_FUNCTION_BLOCK

FUNCTION_BLOCK fbLascoBmin (*Betriebsdauer in Minuten zählen*)
	VAR_INPUT
		Aktiv : BOOL; (*Betriebsmittel Aktiv*)
		sekTick : BOOL; (*Sekundentakt*)
		Minuten : REFERENCE TO USINT; (*Ausgabe Minuten*)
		Reset : BOOL; (*Rücksetzen*)
	END_VAR
	VAR
		Sekunden : USINT;
	END_VAR
END_FUNCTION_BLOCK

FUNCTION_BLOCK fbLascoStdMin (*Angehängte Betriebsdauer von Minuten in Stunden umwandeln*)
	VAR_INPUT
		Minuten : REFERENCE TO USINT; (*Betriebsdauer in Minuten*)
		Stunden : REFERENCE TO UDINT; (*Betriebsdauer in Stunden*)
		Reset : BOOL; (*Rücksetzen*)
	END_VAR
END_FUNCTION_BLOCK

FUNCTION_BLOCK fbLascoSrvcInterv (*Funktionsbaustein für Serviceintervalle*)
	VAR_INPUT
		Aktiv : BOOL; (*Bauteil aktiv*)
		Tick : BOOL; (*Taktfrequenz*)
		SrvcIntervall : UDINT; (*Serviceintervall*)
		ZeitBisSrvc : REFERENCE TO UDINT; (*Verbleibende Zeit bis zum Service*)
		SrvcReset : BOOL; (*Servicemeldung zurücksetzen*)
	END_VAR
	VAR_OUTPUT
		SrvcErforderl : BOOL; (*Meldung Service erforderlich*)
	END_VAR
	VAR
		zzEdge00000 : BOOL;
	END_VAR
END_FUNCTION_BLOCK

FUNCTION_BLOCK fbLascoBrStfLst (*Berechnung der Brennstoffleistung*)
	VAR_INPUT
		sekTick : BOOL; (*Sekundentakt*)
		LeistungAkt : REAL; (*Aktuelle Leistung in kW*)
		Leistung_MWh : REFERENCE TO UDINT; (*Erbrachte Brennstoffleistung in MWh*)
		Leistung_kWh : REFERENCE TO REAL; (*Erbrachte Brennstoffleistung in kWh*)
		Reset : BOOL; (*Rücksetzen*)
	END_VAR
	VAR
		LeistungSek : REAL;
	END_VAR
END_FUNCTION_BLOCK

FUNCTION_BLOCK fbLascoWoPrg (*Wochenprogramm*)
	VAR_INPUT
		Freigabe : BOOL; (*Freigabe *)
		WoPrg : ARRAY[0..7] OF WoPrg_type; (*Feld Wochenprogramm (Heizzeiten pro Wochentag)*)
	END_VAR
	VAR_OUTPUT
		WoPrgFreigabe : BOOL; (*Ausgang Freigabe Wochenprogramm*)
		WoTag : USINT;
	END_VAR
	VAR
		EUhr : fbLascoEUhr;
		StartZeit_1 : REAL;
		StopZeit_1 : REAL;
		StartZeit_2 : REAL;
		StopZeit_2 : REAL;
		AktZeit : REAL;
		FreigabeZeit_1 : BOOL;
		FreigabeZeit_2 : BOOL;
	END_VAR
END_FUNCTION_BLOCK

FUNCTION_BLOCK fbLascoDrzuebw (*Drehzahlüberwachung eines Motors*)
	VAR_INPUT
		Motor : BOOL; (*Motor läuft*)
		Impuls : BOOL; (*Drehimpuls*)
		Tick : BOOL; (*Takt*)
		Zeit : REAL; (*max. Dauer Stillstand*)
		Quit : BOOL; (*Fehlerquittierung*)
	END_VAR
	VAR_OUTPUT
		Fehler : BOOL; (*Fehlerausgang*)
	END_VAR
	VAR
		nextStep : USINT;
		curStep : USINT;
		ElapsedTime : REAL;
	END_VAR
END_FUNCTION_BLOCK

FUNCTION_BLOCK fbLascoFehl (*Fehlerverzögerung und Quittierungsverhalten*)
	VAR_INPUT
		FehlerIn : BOOL; (*Fehlereingang*)
		VerzZeit : REAL; (*Verzögerungszeit*)
		Quit : BOOL; (*Fehlerquittierung*)
		Tick : BOOL; (*Taktfrequenz*)
		Mode : USINT; (*0= Fehlerdominant, nur rücksetzbar wenn kein Fehlereingang/1= Quittierdominant/2= Quittierdominant, keine Selbsthaltung /3= Keine Quittierung, keine Selbsthaltung /4= Selbstquittierung*)
	END_VAR
	VAR_OUTPUT
		FehlerOut : BOOL; (*Fehlerausgang*)
	END_VAR
	VAR
		Counter : REAL;
	END_VAR
END_FUNCTION_BLOCK

FUNCTION_BLOCK fbLascoFept (*Fehlergenerierung PT100- Eingang*)
	VAR_INPUT
		IN : REAL; (*PT100- Wert*)
		Quit : BOOL; (*Fehlerquittierung*)
		Enable : BOOL; (*Freigabe*)
		Tick : BOOL; (*Taktfrequenz*)
		VerzZeit : REAL; (*Fehlerverzögerung*)
	END_VAR
	VAR_OUTPUT
		Q : BOOL; (*Fehlerausgang*)
	END_VAR
	VAR
		Counter : REAL;
	END_VAR
END_FUNCTION_BLOCK

FUNCTION_BLOCK fbLascoPuge (*Pulsgenerator*)
	VAR_INPUT
		StartMitPuls : BOOL; (*Mit Puls Starten*)
		StartMitPause : BOOL; (*Mit Pause Starten*)
		Tick : BOOL; (*Taktfrequeunz*)
		ZeitPuls : REAL; (*Pulszeit*)
		ZeitPause : REAL; (*Pausenzeit*)
		Reset : BOOL; (*Reset Pulszeit*)
	END_VAR
	VAR_OUTPUT
		PulsQ : BOOL; (*Puls*)
		PauseQ : BOOL; (*Pause*)
		RestzeitPuls : REAL; (*Restliche Pulszeit*)
		RestzeitPause : REAL; (*Restliche Pausenzeit*)
	END_VAR
	VAR
		currStep : USINT;
		CounterPuls : REAL;
		CounterPause : REAL;
		nextStep : USINT;
	END_VAR
END_FUNCTION_BLOCK

FUNCTION_BLOCK fbLascoLstgStell (*Leistungssteller*)
	VAR_INPUT
		Enable : BOOL; (*Freigabe*)
		GesLeistungMin : REAL; (*Minimale Gesamtleistung*)
		GesLeistungMax : REAL; (*Maximale Gesamtleistung*)
		EinschubPulsMin : REAL; (*Minimale Pulszeit Einschubschnecke*)
		EinschubPulsMax : REAL; (*Maximale Pulszeit Einschubschnecke*)
		SaugzugDrehzMin : REAL; (*Minimale Drehzahl Saugzuggebläse*)
		SaugzugDrehzMax : REAL; (*Maximale Drehzahl Saugzuggebläse*)
		PrimaerStellMin : REAL; (*Minimale Stellung Primärluftklappe*)
		PrimaerStellMax : REAL; (*Maximale Stellung Primärklappe*)
		EinschubPauseMin : REAL; (*Minimale Pulszeit Einschubschnecke*)
		EinschubPauseMax : REAL; (*Maximale Pulszeit Einschubschnecke*)
		SekundaerStellMin : REAL; (*Minimale Stellung Sekundärklappe*)
		SekundaerStellMax : REAL; (*Maximale Stellung Sekundärklappe*)
		GesLeistungSoll : REAL; (*Leistung Sollwert*)
		RostPulsMin : REAL;
		RostPulsMax : REAL;
		RostPauseMin : REAL;
		RostPauseMax : REAL;
		ReziStellMin : REAL;
		ReziStellMax : REAL;
	END_VAR
	VAR_OUTPUT
		EinschubPulsSoll : UDINT; (*Stellgröße Puls Einschub*)
		EinschubPauseSoll : UDINT; (*Stellgröße Pause Einschub*)
		PrimaerStellSoll : REAL; (*Stellgröße Primärklappe*)
		SekundaerStellSoll : REAL; (*Stellgröße Sekundärklappe*)
		SaugzugDrehzSoll : REAL; (*Stellgröße Saugzuggebläse*)
		ReziStellSoll : REAL;
		RostPulsSoll : UDINT;
		RostPauseSoll : UDINT;
	END_VAR
	VAR
		ScalDrehzSaugzug : LCRLimScal;
		ScalStellPrimaer : LCRLimScal;
		ScalStellSekundaer : LCRLimScal;
		ScalPulsEinschub : LCRLimScal;
		ScalPauseEinschub : LCRLimScal;
		ScalPulsRost : LCRLimScal;
		ScalPauseRost : LCRLimScal;
		ScalStellRezi : LCRLimScal;
	END_VAR
END_FUNCTION_BLOCK

FUNCTION_BLOCK fbLascoLstRamp (*Rampenfunktion, Leistungsanstieg pro Minute*) (*$GROUP=Lasco,$CAT=Warmluftofen,$GROUPICON=LD_user.png,$CATICON=LD_basic.png*)
	VAR_INPUT
		Enable : BOOL; (*Freigabe*)
		LeistungStart : REAL; (*Leistung Out bei Start der Funktion*)
		LeistungSoll : REAL; (*Leistungsvorgabe*)
		sekTick : BOOL; (*Sekundentakt*)
		AnstiegProMinute : REAL; (*Leistungsanstieg pro Minute*)
		Pause : BOOL;
		LeistungOut : REFERENCE TO REAL;
	END_VAR
	VAR_OUTPUT
		Fertig : BOOL; (*Meldung Fertig*)
	END_VAR
	VAR
		AnstiegProSekunde : REAL;
		zzEdge00000 : BOOL;
	END_VAR
END_FUNCTION_BLOCK

FUNCTION_BLOCK fbLascoZund (*Funktionsblock Zündgebläse*)
	VAR_INPUT
		Freigabe : BOOL; (*Freigabe Zündung*)
		IstTemp : REAL; (*Ist- Temperatur Brennraum*)
		SollTemp : REAL; (*Soll- Temperatur Brennraum*)
		Zuendzeit : REAL; (*Max. Zündzeit*)
		Nachlaufzeit : REAL; (*Nachlaufzeit Zündgebläse*)
		Tick : BOOL; (*Taktfrequenz für Zeitglieder*)
	END_VAR
	VAR_OUTPUT
		Zuendspule : BOOL; (*Ausgang Zündspule*)
		ZuendungOK : BOOL; (*Meldung Zündung OK*)
		ZuendungFehler : BOOL; (*Fehlermeldung Zündung*)
		Zuendgeblaese : BOOL; (*Ausgang Zündgebläse*)
	END_VAR
	VAR
		TON_Zuendzeit : fbLascoTON;
		TOF_Nachlaufzeit : fbLascoTOF;
	END_VAR
END_FUNCTION_BLOCK

FUNCTION_BLOCK fbLascoFU (*Ansteuerung Frequenzumrichter*)
	VAR_INPUT
		Freigabe : BOOL; (*Umrichter Freigabe*)
		SollDrehzahl : REAL; (*Drehzahlvorgabe*)
		AnsprechZeitFU : REAL; (*Max. Ansprechverzögerung Betriebsmeldung*)
		BetrMldg : BOOL; (*Betriebsmeldung*)
		RampeUpSek : REAL; (*Rampenzeit Drehzahlerhöhung (sek)*)
		RampeDownSek : REAL; (*Rampenzeit Drehzahlverminderung (sek)*)
		Reset : BOOL; (*Fehler- Reset*)
		Tick : BOOL; (*Taktfrequenz Zeitglieder*)
		MaxDrehzahl : REAL; (*Maximale Drehzahl Umrichter*)
		MinDrehzahl : REAL; (*Minimale Drehzahl Umrichter*)
	END_VAR
	VAR_OUTPUT
		BetriebFU : BOOL; (*Umrichter Betrieb*)
		StoerungFU : BOOL; (*Fehlerausgang*)
		DrehzahlFU : REAL; (*Drehzahlvorgabe*)
	END_VAR
	VAR
		TON_Betriebsmeldung : fbLascoTON;
		zzEdge00000 : BOOL;
		zzEdge00001 : BOOL;
		zzEdge00002 : BOOL;
		InitDone : BOOL;
		ResetDone : BOOL;
		LCRRamp_0 : LCRRamp;
		RampDownMillis : DINT;
		RampUpMillis : DINT;
		IstDrehzahl : REAL;
		Init : BOOL;
		zzEdge00003 : BOOL;
	END_VAR
END_FUNCTION_BLOCK

FUNCTION_BLOCK fbLascoZweiPunktAchse (*Ansteuerung Zweipunktachse*)
	VAR_INPUT
		Freigabe : BOOL; (*Freigabe *)
		Vor : BOOL; (*Befehl Vorwärts*)
		Zurueck : BOOL; (*Befehl Rückwärts*)
		AnsprechZeit : REAL; (*Ansprechverzögerung*)
		MinLaufZeit : REAL; (*Nachlaufzeit*)
		Stoerung : BOOL; (*Störungseingang*)
		ESVor : BOOL; (*Endlage Vorwärtsbewegung*)
		ESZurueck : BOOL; (*Endlage Rückwärtsbewegung*)
		Tick : BOOL; (*Taktfrequenz*)
	END_VAR
	VAR_OUTPUT
		Motor_Vor : BOOL; (*Ausgang Vorwärts*)
		Motor_Zurueck : BOOL; (*Ausgang Rückwärts*)
		Fehler : BOOL; (*Fehlerausgang*)
	END_VAR
	VAR
		TON_Ansprechzeit : fbLascoTON;
		TOF_Laufzeit : fbLascoTOF;
		loc_Vor : BOOL;
		TON_AnsprechzeitZurueck : fbLascoTON;
		TOF_LaufzeitZurueck : fbLascoTOF;
		loc_Zurueck : BOOL;
	END_VAR
END_FUNCTION_BLOCK

FUNCTION_BLOCK fbLascoStellachse (*Ansteuerung Stellachsen*)
	VAR_INPUT
		Freigabe : BOOL; (*Achse Freigabe*)
		Stoerung : BOOL; (*Fehlereingang*)
		SollStellung : REAL; (*Vorgabe Stellung*)
		IstStellung : REAL; (*Istwert Stellung*)
		EsVor : BOOL; (*Endlage Auf-Bewegung*)
		Hysterese : REAL; (*Hysterese zw. Soll- und Iststellung*)
		EsZurueck : BOOL; (*Endlage Zu-Bewegung*)
	END_VAR
	VAR_OUTPUT
		MotorVor : BOOL; (*Ausgang Motor Vor*)
		MotorZurueck : BOOL; (*Ausgang Motor Zurück*)
		Fehler : BOOL;
	END_VAR
END_FUNCTION_BLOCK

FUNCTION_BLOCK fbLascoStellachseAnalog (*Ansteuerung von analogen Stellachsen*)
	VAR_INPUT
		Freigabe : BOOL; (*Achse Freigabe*)
		SollStellung : REAL; (*Vorgabe Stellung*)
		IstStellung : REAL; (*Istwert Stellung*)
		Hysterese : REAL; (*Hysterse zw. Soll- und Iststellung*)
		EsVor : BOOL; (*Endlage Auf-Bewegung*)
		EsZurueck : BOOL; (*Endlage Zu-Bewegung*)
		Stoerung : BOOL; (*Fehlereingang*)
	END_VAR
	VAR_OUTPUT
		MotorStellung : REAL; (*Ausgang Stellgröße Motor*)
		Fehler : BOOL;
	END_VAR
END_FUNCTION_BLOCK

FUNCTION_BLOCK fbLascoStellachseDigital (*Ansteuerung von Stellachsen ohne Positionsrückmeldung*)
	VAR_INPUT
		Freigabe : BOOL;
		Sollstellung : REAL;
		Referenz : BOOL;
		Oeffnungszeit : REAL;
		Schliesszeit : REAL;
		MinPosition : REAL;
		MaxPosition : REAL;
		MinImpulsdauer : REAL;
		Tick : BOOL; (*Zehntelsekunden- Takt*)
	END_VAR
	VAR_OUTPUT
		ReferenzOk : BOOL;
		MotorAuf : BOOL;
		MotorZu : BOOL;
		ReferenzAktiv : BOOL;
		IstPosition : REAL;
	END_VAR
	VAR
		LCRContinServo_0 : LCRContinServo;
		zzEdge00000 : BOOL;
		WegProZeitAuf : REAL;
		WegProZeitZu : REAL;
		zzEdge00001 : BOOL;
		zzEdge00002 : BOOL;
		zzEdge00003 : BOOL;
	END_VAR
END_FUNCTION_BLOCK

FUNCTION_BLOCK fbLascoWarmluftsteller (*Ansteuerung Warmluftgebläse mit Kühlreduzierung*)
	VAR_INPUT
		Freigabe : BOOL; (*Freigabe*)
		IstTemperatur : REAL; (*Aktuelle Temperatur*)
		GrenzTemperatur : REAL; (*Grenztemperatur*)
		Bezugszeit : REAL; (*Bezugszeit*)
		MinderungDRZ : REAL; (*Drehzahlminderung pro Schritt*)
		Tick : BOOL; (*Taktfrequeunz*)
		WLG1MinDRZ : REAL; (*Gebläse 1 Min. Drehzahl*)
		WLG2MinDRZ : REAL; (*Gebläse 2 Min. Drehzahl*)
		WLG1SollDRZ : REAL; (*Gebläse 1 Soll-Drehzahl*)
		WLG2SollDRZ : REAL; (*Gebläse 2 Soll-Drehzahl*)
	END_VAR
	VAR_OUTPUT
		WLG1DRZStell : REAL; (*Stellgröße Gebläse 1*)
		WLG2DRZStell : REAL; (*Stellgröße Gebläse 2*)
	END_VAR
	VAR
		curState : USINT;
		nextState : USINT;
		stateEntry : BOOL;
		locDrehzahl1 : REAL;
		locDrehzahl2 : REAL;
		TON_WarmluftSteller : fbLascoTON;
	END_VAR
END_FUNCTION_BLOCK

FUNCTION_BLOCK fbLascoFreilauf (*Freilauffunktion für blockierende Motoren*)
	VAR_INPUT
		Freigabe : BOOL; (*Funktion Freigabe*)
		Tick : BOOL; (*Taktfrequenz*)
		Stehzeit : REAL; (*Max. Stehzeit des Motors*)
		Impuls : BOOL; (*Drehimpuls*)
		VerzFreilauf : REAL; (*Verzögerungszeit zw. Richtungswechseln*)
		Freilaufzeit : REAL; (*Freilaufzeit*)
		MaxVersuche : INT; (*Max. Freiläufe pro Minute*)
		Quit : BOOL; (*Fehlerquittierung*)
	END_VAR
	VAR_OUTPUT
		MotorVor : BOOL; (*Freigabe Motor Vorwärts*)
		MotorZurueck : BOOL; (*Freigabe Motor Rückwärts*)
		Fehler : BOOL;
	END_VAR
	VAR
		curStep : USINT;
		nextStep : USINT;
		stateEntry : BOOL;
		DRZWaechter : fbLascoDrzuebw;
		TON_VerzRW : fbLascoTON;
		TON_Freilaufzeit : fbLascoTON;
		CounterVersuche : INT;
		TON_ResetCounter : fbLascoTON;
	END_VAR
END_FUNCTION_BLOCK

FUNCTION_BLOCK fbLascoFuellst (*Überwachung von Fuellstandssensoren*)
	VAR_INPUT
		Fuellstand : BOOL;
		EinschubEin : BOOL;
		Quit : BOOL;
		Tick : BOOL;
		VerzZeit : REAL;
	END_VAR
	VAR_OUTPUT
		Fehler : BOOL;
	END_VAR
	VAR
		cKeineFlankeFs : UDINT;
		zzEdge00000 : BOOL;
	END_VAR
END_FUNCTION_BLOCK

FUNCTION_BLOCK fbLascoWlg (*Ansteuerung für Warmluftgebläse ohne Drehzahlvorgabe*)
	VAR_INPUT
		Freigabe : BOOL; (*Freigabe*)
		StartBeiTemp : REAL; (*Wenn Ist- Temperatur über diesem Wert -> Gebläse Ein*)
		StopBeiTemp : REAL; (*Wenn Ist- Temperatur unter diesem Wert -> Gebläse Aus*)
		IstTemp : REAL; (*Ist- Temperatur*)
		Stoerung : BOOL; (*Störungseingang*)
	END_VAR
	VAR_OUTPUT
		GeblaeseEin : BOOL; (*Ansteuerung Gebläse*)
		Fehler : BOOL; (*Fehlerausgang*)
	END_VAR
END_FUNCTION_BLOCK

FUNCTION_BLOCK fbLascoBsk (*Funktionsbaustein zur Ansteuerung von federrückgestellten Klappenantrieben*) (*$GROUP=Anwender*)
	VAR_INPUT
		Freigabe : BOOL; (*Freigabe Funktionsbaustein*)
		Oeffnen : BOOL; (*Befehl Öffnen*)
		KlappeIstOffen : BOOL; (*Eingang Klappe ist Offen*)
		KlappeIstGeschlossen : BOOL; (*Eingang Klappe ist Geschlossen*)
		FahrzeitAuf : UDINT; (*Fahrzeit Klappe Auf [ms]*)
		FahrzeitZu : UDINT; (*Fahrzeit Klappe Zu [ms]*)
		QuitFehler : BOOL; (*Fehlerquittierung*)
		Stoerung : BOOL; (*Eingang Fehler*)
	END_VAR
	VAR_OUTPUT
		KlappeAuf : BOOL; (*Ausgang Klappe Öffnen*)
		Fehler : BOOL; (*Augang Fehler*)
		FehlerFahrzeitAuf : BOOL; (*Ausgang Fehler beim Öffnen*)
		FehlerFahrzeitZu : BOOL; (*Ausgang Fehler beim Schliessen*)
	END_VAR
	VAR
		TON_FahrzeitAuf : TON;
		TON_FahrzeitZu : TON;
		zzEdge00000 : BOOL;
		zzEdge00001 : BOOL;
		zzEdge00002 : BOOL;
		zzEdge00003 : BOOL;
	END_VAR
END_FUNCTION_BLOCK

FUNCTION_BLOCK fbLascoTrend (*Trenderkennung eines Eingangswertes innerhalb einer Zeitspanne (steigend/fallend)*) (*$GROUP=Anwender*)
	VAR_INPUT
		Freigabe : BOOL;
		Eingangswert : REAL;
		Zeitspanne : REAL;
		Tick : BOOL;
		MinAbweichung : REAL; (*Mindest-Abweichung bis eine Tendenz erkannt wird*)
	END_VAR
	VAR_OUTPUT
		TendenzSteigend : BOOL;
		TendenzFallend : BOOL;
	END_VAR
	VAR
		ctZeitspanne : REAL;
		Mittelwert : REAL;
		SummeWert : LREAL;
		MittelwertMEM : REAL;
		Abweichung : REAL;
	END_VAR
END_FUNCTION_BLOCK

FUNCTION_BLOCK fbLascoTimerHand (*Timer mit Hand-Funktionen*) (*$GROUP=Anwender*)
	VAR_INPUT
		Freigabe : BOOL;
		Zeit : REAL;
		Tick : BOOL;
		HandEin : BOOL;
		HandAus : BOOL;
	END_VAR
	VAR_OUTPUT
		Q : BOOL;
	END_VAR
	VAR
		Elapsed : REAL;
	END_VAR
END_FUNCTION_BLOCK

{REDUND_ERROR} {REDUND_UNREPLICABLE} FUNCTION_BLOCK fbLascoPugeV2 (*Puls/Pause-Generator mit Standard-Timern*) (*$GROUP=User,$CAT=User,$GROUPICON=User.png,$CATICON=User.png*)
	VAR_INPUT
		StartMitPuls : {REDUND_UNREPLICABLE} BOOL;
	END_VAR
	VAR
		curStep : {REDUND_UNREPLICABLE} USINT;
		nextStep : {REDUND_UNREPLICABLE} USINT;
		stateEntry : {REDUND_UNREPLICABLE} BOOL;
	END_VAR
	VAR_OUTPUT
		PulsOut : {REDUND_UNREPLICABLE} BOOL;
		PauseOut : {REDUND_UNREPLICABLE} BOOL;
		RestzeitPause : {REDUND_UNREPLICABLE} UDINT;
		RestzeitPuls : {REDUND_UNREPLICABLE} UDINT;
	END_VAR
	VAR_INPUT
		ZeitPuls : {REDUND_UNREPLICABLE} UDINT;
		StartMitPause : {REDUND_UNREPLICABLE} BOOL;
	END_VAR
	VAR
		TON_Schrittzeit : {REDUND_UNREPLICABLE} TON;
	END_VAR
	VAR_INPUT
		ZeitPause : {REDUND_UNREPLICABLE} UDINT;
	END_VAR
END_FUNCTION_BLOCK
```

#### fbLascoEUhr.st - Echtzeituhr auslesen
```iecst
(********************************************************************
 * COPYRIGHT -- LASCO Heu- und Forsttechnik GmbH
 ********************************************************************
 * Library: LascoUtil
 * Datei: fbLascoEUhr.st
 * Autor: Rudolf Lachner
 * Erstellt: 2. April 2013
 ********************************************************************
 * Implementierung der Library LascoUtil
 ********************************************************************)

(* Echtzeituhr auslesen *)
FUNCTION_BLOCK fbLascoEUhr

	IF (Freigabe = TRUE) THEN

		//Echtzeituhr auslesen
		RTC_gettime(ADR(Echtzeit));

		//Datum und Uhrzeit auslesen
		DTGetTime_0.enable	:= TRUE;
		DTGetTime_0();
		DateTime			:= DTGetTime_0.DT1;

		//Zeit als Word bilden
		StdMin		:= (Echtzeit.Stunde * 100) + Echtzeit.Minute;

		//Zeit ausgeben
		Jahr		:= Echtzeit.Jahr;
		Monat		:= Echtzeit.Monat;
		Tag			:= Echtzeit.Tag;
		WoTag		:= Echtzeit.WoTag;
		Stunde		:= Echtzeit.Stunde;
		Minute		:= Echtzeit.Minute;
		Sekunde		:= Echtzeit.Sekunde;
		Milli		:= Echtzeit.Milli;
		Mikro		:= Echtzeit.Mikro;

	ELSE

		Jahr		:= 0;
		Monat		:= 0;
		Tag			:= 0;
		WoTag		:= 0;
		Stunde		:= 0;
		Minute		:= 0;
		Sekunde		:= 0;
		Milli		:= 0;
		Mikro		:= 0;
		StdMin		:= 0;

	END_IF

END_FUNCTION_BLOCK
```

#### fbLascoTON.st - Einschaltverzögerung
```iecst
(********************************************************************
 * COPYRIGHT -- LASCO Heu- und Forsttechnik GmbH
 ********************************************************************
 * Library: LascoUtil
 * Datei: fbLascoTON.st
 * Autor: Rudolf Lachner
 * Erstellt: 28. März 2013
 ********************************************************************
 * Implementierung der Library LascoUtil
 ********************************************************************)

(* Einschaltverzögerung *)
FUNCTION_BLOCK fbLascoTON

	IF (NOT IN) THEN
		Elapsed	:= 0;
		Q		:= FALSE;
	ELSIF (Elapsed	>= Zeit) THEN
		Q		:= TRUE;
	ELSE
		Elapsed	:= Elapsed + Tick;
		Q		:= FALSE;
	END_IF

END_FUNCTION_BLOCK
```

#### fbLascoTOF.st - Ausschaltverzögerung
```iecst
(********************************************************************
 * COPYRIGHT -- LASCO Heu- und Forsttechnik GmbH
 ********************************************************************
 * Library: LascoUtil
 * Datei: fbLascoTOF.st
 * Autor: Rudolf Lachner
 * Erstellt: 28. März 2013
 ********************************************************************
 * Implementierung der Library LascoUtil
 ********************************************************************)

(* Ausschaltverzögerung *)
FUNCTION_BLOCK fbLascoTOF

	IF (Reset) THEN
		Q		:= FALSE;
		Elapsed	:= 0;

	ELSIF (IN) THEN
		Q		:= TRUE;
		Elapsed	:= 0;

	ELSIF (Q AND NOT IN) THEN

		IF (Elapsed < Zeit) THEN
			Elapsed	:= Elapsed + Tick;
		ELSE
			Q		:= FALSE;
			Elapsed	:= 0;
		END_IF

	END_IF

END_FUNCTION_BLOCK
```

#### fbLascoTOG.st - Toggle- Funktion
```iecst
(********************************************************************
 * COPYRIGHT -- LASCO Heu- und Forsttechnik GmbH
 ********************************************************************
 * Library: LascoUtil
 * Datei: fbLascoTOG.st
 * Autor: Rudolf Lachner
 * Erstellt: 28. März 2013
 ********************************************************************
 * Implementierung der Library LascoUtil
 ********************************************************************)

(* Toggle- Funktion *)
FUNCTION_BLOCK fbLascoTOG

	IF Reset THEN
		Q     	:= FALSE;
		ToggImp := FALSE;

	ELSIF (NOT IN) THEN
		ToggImp := FALSE;

	ELSIF (IN AND NOT ToggImp AND NOT Q) THEN
		Q     	:= TRUE;
		ToggImp := TRUE;

	ELSIF (IN AND NOT ToggImp AND Q) THEN
		Q     	:= FALSE;
		ToggImp := TRUE;
	END_IF

END_FUNCTION_BLOCK
```

#### funLascoMinss.st
```iecst
(********************************************************************
 * COPYRIGHT -- LASCO Heu- und Forsttechnik GmbH
 ********************************************************************
 * Library: LascoUtil
 * Datei: funLascoMinss.st
 * Autor: Rudolf Lachner
 * Erstellt: 28. März 2013
 ********************************************************************
 * Implementierung der Library LascoUtil
 ********************************************************************)

(* Wert in Minuten und Sekunden umwandeln*)
FUNCTION funLascoMinss

	//Eine Eingabe von 5.30 m.ss ergibt dadurch 5 Minunten und 30 Sekunden;

	funLascoMinss := ((IN / 100) * 60) + (IN - (IN / 100) * 100);

END_FUNCTION
```

#### fbLascoZdxx.st - Tickausgabe bei Zustandsänderung des Einganges
```iecst
(********************************************************************
 * COPYRIGHT -- LASCO Heu- und Forsttechnik GmbH
 ********************************************************************
 * Library: LascoUtil
 * Datei: fbLascoZdxx.st
 * Autor: Rudolf Lachner
 * Erstellt: 27. März 2013
 ********************************************************************
 * Implementierung der Library LascoUtil
 ********************************************************************)

(* Tickausgabe bei Zustandsänderung des Einganges *)
FUNCTION_BLOCK fbLascoZdxx

	IF (IN <> MEM) THEN
		MEM	:= IN;
		Q	:= TRUE;
	ELSE
		Q	:= FALSE;
	END_IF

END_FUNCTION_BLOCK
```

#### fbLascoZbFrg.st - Zeitfenster Freigabe
```iecst
(********************************************************************
 * COPYRIGHT -- LASCO Heu- und Forsttechnik GmbH
 ********************************************************************
 * Library: LascoUtil
 * Datei: fbLascoZbFrg.st
 * Autor: Rudolf Lachner
 * Erstellt: 3. April 2013
 ********************************************************************
 * Implementierung der Library LascoUtil
 ********************************************************************)

(* Zeitfenster Freigabe *)
FUNCTION_BLOCK fbLascoZbFrg

	//Akutelle Uhrzeit auslesen
	EUhr(Freigabe := TRUE);
	AktZeit	:= INT_TO_REAL(EUhr.StdMin);

	IF (Freigabe = TRUE) THEN

		FreigZeitfenster	:= FALSE;
		IF (StartZeit > StoppZeit) THEN
			IF (AktZeit >= StartZeit) OR (AktZeit < StoppZeit) THEN
				FreigZeitfenster 	:= TRUE;
			END_IF
		ELSE
			IF (AktZeit >= StartZeit) AND (AktZeit < StoppZeit) THEN
				FreigZeitfenster	:= TRUE;
			END_IF
		END_IF

	ELSE
		FreigZeitfenster	:= FALSE;
	END_IF

END_FUNCTION_BLOCK
```

#### fbLascoBstd.st - Betriebsstundenzähler auf Minutenbasis
```iecst
(********************************************************************
 * COPYRIGHT -- LASCO Heu- und Forsttechnik GmbH
 ********************************************************************
 * Library: LascoUtil
 * Datei: fbLascoBstd.st
 * Autor: Rudolf Lachner
 * Erstellt: 27. März 2013
 ********************************************************************
 * Implementierung der Library LascoUtil
 ********************************************************************)

(* Betriebsstundenzähler auf Minutenbasis *)
FUNCTION_BLOCK fbLascoBstd

	IF (Aktiv AND minTick) THEN

		IF Minuten < 59 THEN
			Minuten	:= Minuten + 1;
		ELSE
			Stunden	:= Stunden + 1;
			Minuten	:= 0;
		END_IF

	END_IF

	IF (Reset) THEN
		Minuten	:= 0;
		Stunden	:= 0;
	END_IF

END_FUNCTION_BLOCK
```

#### fbLascoWoPrg.st - Wochenprogramm
```iecst
(********************************************************************
 * COPYRIGHT -- LASCO Heu- und Forsttechnik GmbH
 ********************************************************************
 * Library: LascoUtil
 * Datei: fbLascoWoPrg.st
 * Autor: Rudolf Lachner
 * Erstellt: 2. April 2013
 ********************************************************************
 * Implementierung der Library LascoUtil
 ********************************************************************)

(* Wochenprogramm *)
FUNCTION_BLOCK fbLascoWoPrg

	//Akutelle Uhrzeit auslesen
	EUhr(Freigabe := TRUE);
	WoTag	:= EUhr.WoTag;
	AktZeit	:= INT_TO_REAL(EUhr.StdMin);

	//Zeitfenster auswerten
	//=====================

	//Heizzeit 1
	StartZeit_1	:= (WoPrg[WoTag].HZ1_Std_Ein * 100) + WoPrg[WoTag].HZ1_Min_Ein;
	StopZeit_1	:= (WoPrg[WoTag].HZ1_Std_Aus * 100) + WoPrg[WoTag].HZ1_Min_Aus;

	FreigabeZeit_1	:= FALSE;
	IF (StartZeit_1 > StopZeit_1) THEN
		IF (AktZeit >= StartZeit_1) OR (AktZeit < StopZeit_1) THEN
			FreigabeZeit_1 	:= TRUE;
		END_IF
	ELSE
		IF (AktZeit >= StartZeit_1) AND (AktZeit < StopZeit_1) THEN
			FreigabeZeit_1	:= TRUE;
		END_IF
	END_IF

	//Heizzeit 2
	StartZeit_2	:= (WoPrg[WoTag].HZ2_Std_Ein * 100) + WoPrg[WoTag].HZ2_Min_Ein;
	StopZeit_2	:= (WoPrg[WoTag].HZ2_Std_Aus * 100) + WoPrg[WoTag].HZ2_Min_Aus;

	FreigabeZeit_2	:= FALSE;
	IF (StartZeit_2 > StopZeit_2) THEN
		IF (AktZeit >= StartZeit_2) OR (AktZeit < StopZeit_2) THEN
			FreigabeZeit_2 	:= TRUE;
		END_IF
	ELSE
		IF (AktZeit >= StartZeit_2) AND (AktZeit < StopZeit_2) THEN
			FreigabeZeit_2	:= TRUE;
		END_IF
	END_IF

	//Freigabe generieren
	IF (Freigabe= TRUE) THEN

		WoPrgFreigabe	:= (FreigabeZeit_1 AND WoPrg[WoTag].HZ1_Enable) OR (FreigabeZeit_2 AND WoPrg[WoTag].HZ2_Enable);
	ELSE

		WoPrgFreigabe	:= FALSE;

	END_IF

END_FUNCTION_BLOCK
```

#### fbLascoDrzuebw.st - Drehzahlüberwachung eines Motors
```iecst
(********************************************************************
 * COPYRIGHT -- LASCO Heu- und Forsttechnik GmbH
 ********************************************************************
 * Library: LascoUtil
 * Datei: fbLascoDrzuebw.st
 * Autor: Rudolf Lachner
 * Erstellt: 27. März 2013
 ********************************************************************
 * Implementierung der Library LascoUtil
 ********************************************************************)

(* Drehzahlüberwachung eines Motors *)
FUNCTION_BLOCK fbLascoDrzuebw

	//Schrittschaltwerk Impulsüberwachung
	//===================================

	curStep	:= nextStep;

	CASE curStep OF

		//**************************************************************************************************************************************************************************************
		0://MOTOR AUS

			//*** state during ***
			Fehler := FALSE;

			//*** state exit ***

			//Motor ein, kein Impuls
			IF (Motor) AND (NOT Impuls) THEN
				nextStep	:= 1;

			//Motor ein, Impuls
			ELSIF (Motor) AND (Impuls) THEN
				nextStep	:= 2;
			END_IF

		//*********************************************************************************************************************************************************
		1://KEIN IMPULS

			//*** state during ***
			Fehler 		:= FALSE;
			ElapsedTime	:= ElapsedTime + Tick;

			//*** state exit ***

			//Überwachungszeit abgelaufen
			IF (ElapsedTime >= Zeit) THEN
				nextStep	:= 255;

			//Impuls
			ELSIF (Impuls) THEN
				ElapsedTime	:= 0;
				nextStep	:= 2;

			//Motor AUS
			ELSIF (NOT Motor) THEN
				ElapsedTime	:= 0;
				nextStep	:= 0;
			END_IF

		//*******************************************************************************************************************************************************
		2://IMPULS

			//*** state during ***
			Fehler 		:= FALSE;
			ElapsedTime	:= ElapsedTime + Tick;

			//*** state exit ***

			//Überwachungszeit abgelaufen
			IF (ElapsedTime >= Zeit) THEN
				nextStep	:= 255;

			//Kein Impuls
			ELSIF (NOT Impuls) THEN
				ElapsedTime	:= 0;
				nextStep	:= 1;

			//Motor AUS
			ELSIF (NOT Motor) THEN
				ElapsedTime	:= 0;
				nextStep	:= 0;
			END_IF

		//*******************************************************************************************************************************************************************
		255://FEHLER

			//*** state during ***
			Fehler 		:= TRUE;
			ElapsedTime	:= 0;

			//*** state exit ***

			//Fehler quittiert
			IF (Quit) THEN
				nextStep	:= 0;
			END_IF

	END_CASE

END_FUNCTION_BLOCK
```

#### fbLascoFehl.st - Fehlerverzögerung und Quittierungsverhalten
```iecst
(********************************************************************
 * COPYRIGHT -- LASCO Heu- und Forsttechnik GmbH
 ********************************************************************
 * Library: LascoUtil
 * Datei: fbLascoFehl.st
 * Autor: Rudolf Lachner
 * Erstellt: 27. März 2013
 ********************************************************************
 * Implementierung der Library LascoUtil
 ********************************************************************)

(* Fehlerverzögerung und Quittierungsverhalten *)
FUNCTION_BLOCK fbLascoFehl

	//Fehlerdominant + Selbsthaltung
	IF (Mode = 0) THEN

		IF (Quit AND NOT FehlerIn) OR (NOT FehlerIn AND NOT FehlerOut) THEN
			Counter		:= 0;
			FehlerOut	:= FALSE;
		ELSIF (Counter < VerzZeit) AND (NOT FehlerOut) THEN
			Counter		:= Counter + Tick;
		ELSE
			FehlerOut	:= TRUE;
		END_IF

	//Quittierdominant + Selbsthaltung
	ELSIF (Mode = 1) THEN

		IF (Quit) OR (NOT FehlerIn AND NOT FehlerOut) THEN
			Counter		:= 0;
			FehlerOut	:= FALSE;
		ELSIF (Counter < VerzZeit) AND (NOT FehlerOut) THEN
			Counter		:= Counter + Tick;
		ELSE
			FehlerOut	:= TRUE;
		END_IF

	//Quittierdominamt, keine Selbsthaltung
	ELSIF (Mode = 2) THEN

		IF (Quit) OR (NOT FehlerIn) THEN
			Counter		:= 0;
			FehlerOut	:= FALSE;
		ELSIF (Counter < VerzZeit) AND (NOT FehlerOut) THEN
			Counter		:= Counter + Tick;
		ELSE
			FehlerOut	:= TRUE;
		END_IF

	//Keine Quittierung, keine Selbsthaltung
	ELSIF (Mode = 3) THEN

		IF (NOT FehlerIn) THEN
			Counter		:= 0;
			FehlerOut	:= FALSE;
		ELSIF (Counter < VerzZeit) AND (NOT FehlerOut) THEN
			Counter		:= Counter + Tick;
		ELSE
			FehlerOut	:= TRUE;
		END_IF

	//Fehlerdominant, Selbstquittierung
	ELSIF (Mode = 4) THEN

		IF (Quit AND FehlerOut) OR (NOT FehlerIn) THEN
			Counter		:= 0;
			FehlerOut	:= FALSE;
		ELSIF (Counter < VerzZeit) AND (NOT FehlerOut) THEN
			Counter		:= Counter + Tick;
		ELSE
			FehlerOut	:= TRUE;
		END_IF

	END_IF

END_FUNCTION_BLOCK
```

#### fbLascoFept.st - Fehlergenerierung PT100- Eingang
```iecst
(********************************************************************
 * COPYRIGHT -- LASCO Heu- und Forsttechnik GmbH
 ********************************************************************
 * Library: LascoUtil
 * Datei: fbLascoFept.st
 * Autor: Rudolf Lachner
 * Erstellt: 28. März 2013
 ********************************************************************
 * Implementierung der Library LascoUtil
 ********************************************************************)

(* Fehlergenerierung PT100- Eingang *)
FUNCTION_BLOCK fbLascoFept

	//Wert im normalen Bereich UND Quittierung
	IF (Quit) AND (IN < 750) AND (IN > -50) THEN
		Q		:= FALSE;
		Counter	:= 0;

	//Fehler anstehend, Quittierung oder keine Freigabe
	ELSIF (Quit AND Q) OR (NOT Enable) THEN
		Q		:= FALSE;
		Counter	:= 0;

	//Zeit überschritten
	ELSIF (Counter >= VerzZeit) THEN
		Q		:= TRUE;

	//Wert außerhalb des normalen Bereiches
	ELSIF (IN > 750) OR (IN < -50) THEN
		Counter	:= Counter + Tick;
	ELSE
		Counter := 0;
	END_IF

END_FUNCTION_BLOCK
```

#### fbLascoPuge.st - Pulsgenerator
```iecst
(********************************************************************
 * COPYRIGHT -- LASCO Heu- und Forsttechnik GmbH
 ********************************************************************
 * Library: LascoUtil
 * Datei: fbLascoPuge.st
 * Autor: Rudolf Lachner
 * Erstellt: 28. März 2013
 ********************************************************************
 * Implementierung der Library LascoUtil
 ********************************************************************)

(* Pulsgenerator *)
FUNCTION_BLOCK fbLascoPuge

	//Schrittschaltwerk Pulsgenerator
	//===============================

	currStep	:= nextStep;

	CASE currStep OF

		//*******************************************************************************************************************************************************************************
		0://AUSWAHL

			//*** state during ***
			PulsQ			:= FALSE;
			PauseQ			:= FALSE;

			CounterPuls		:= 0;
			CounterPause	:= 0;
			RestzeitPause	:= 0;
			RestzeitPuls	:= 0;

			//*** state exit ***
			IF (StartMitPuls) AND (ZeitPuls <> 0) THEN
				nextStep	:= 2;
			ELSIF (StartMitPause) THEN
				nextStep	:= 1;
			END_IF

		//***********************************************************************************************************************************************************************************
		1://PAUSE

			//*** state during ***
			PulsQ	:= FALSE;
			PauseQ	:= TRUE;

			CounterPause	:= CounterPause + Tick;
			RestzeitPause	:= ZeitPause - CounterPause;
			RestzeitPuls	:= 0;

			//*** state exit ***
			IF ((NOT StartMitPause AND NOT StartMitPuls)) OR (ZeitPuls = 0) THEN
				nextStep	:= 0;
			ELSIF (CounterPause >= ZeitPause) THEN
				CounterPause	:= 0;
				nextStep		:= 2;
			END_IF

		//************************************************************************************************************************************************************************************************
		2://PULS

			//*** state during ***
			PulsQ		:= TRUE;
			PauseQ		:= FALSE;

			CounterPuls		:= CounterPuls + Tick;
			RestzeitPause	:= 0;
			RestzeitPuls	:= ZeitPuls - CounterPuls;

			//*** state exit ***
			IF (CounterPuls >= ZeitPuls) OR (Reset) THEN
				CounterPuls	:= 0;
				nextStep	:= 1;
			END_IF

	END_CASE

END_FUNCTION_BLOCK
```

#### fbLascoLstgStell.st - Leistungssteller
```iecst
(********************************************************************
 * COPYRIGHT -- LASCO Heu- und Forsttechnik GmbH
 ********************************************************************
 * Library: LascoUtil
 * Datei: fbLascoLstgStell.st
 * Autor: Rudolf Lachner
 * Erstellt: 28. März 2013
 ********************************************************************
 * Implementierung der Library LascoUtil
 ********************************************************************)

(* Leistungssteller *)
FUNCTION_BLOCK fbLascoLstgStell

	IF (Enable) THEN

		//Soll-Drehzahl Saugzug bestimmen
		ScalDrehzSaugzug.x		:= GesLeistungSoll;
		ScalDrehzSaugzug.x1		:= GesLeistungMin;
		ScalDrehzSaugzug.x2		:= GesLeistungMax;
		ScalDrehzSaugzug.y1		:= SaugzugDrehzMin;
		ScalDrehzSaugzug.y2		:= SaugzugDrehzMax;
		ScalDrehzSaugzug();

		//Sollstellung Primärklappe
		ScalStellPrimaer.x		:= GesLeistungSoll;
		ScalStellPrimaer.x1		:= GesLeistungMin;
		ScalStellPrimaer.x2		:= GesLeistungMax;
		ScalStellPrimaer.y1		:= PrimaerStellMin;
		ScalStellPrimaer.y2		:= PrimaerStellMax;
		ScalStellPrimaer();

		//Sollstellung Sekundärklappe
		ScalStellSekundaer.x	:= GesLeistungSoll;
		ScalStellSekundaer.x1	:= GesLeistungMin;
		ScalStellSekundaer.x2	:= GesLeistungMax;
		ScalStellSekundaer.y1	:= SekundaerStellMin;
		ScalStellSekundaer.y2	:= SekundaerStellMax;
		ScalStellSekundaer();

		//Sollstellung Reziklappe
		ScalStellRezi.x			:= GesLeistungSoll;
		ScalStellRezi.x1		:= GesLeistungMin;
		ScalStellRezi.x2		:= GesLeistungMax;
		ScalStellRezi.y1		:= ReziStellMin;
		ScalStellRezi.y2		:= ReziStellMax;
		ScalStellRezi();

		//Pulszeit Einschub
		ScalPulsEinschub.x		:= GesLeistungSoll;
		ScalPulsEinschub.x1		:= GesLeistungMin;
		ScalPulsEinschub.x2		:= GesLeistungMax;
		ScalPulsEinschub.y1		:= EinschubPulsMin;
		ScalPulsEinschub.y2		:= EinschubPulsMax;
		ScalPulsEinschub();

		//Pausenzeit Einschub
		ScalPauseEinschub.x		:= GesLeistungSoll;
		ScalPauseEinschub.x1	:= GesLeistungMin;
		ScalPauseEinschub.x2	:= GesLeistungMax;
		ScalPauseEinschub.y1	:= EinschubPauseMin;
		ScalPauseEinschub.y2	:= EinschubPauseMax;
		ScalPauseEinschub();

		//Pulszeit Rost
		ScalPulsRost.x			:= GesLeistungSoll;
		ScalPulsRost.x1			:= GesLeistungMin;
		ScalPulsRost.x2			:= GesLeistungMax;
		ScalPulsRost.y1			:= RostPulsMin;
		ScalPulsRost.y2			:= RostPulsMax;
		ScalPulsRost();

		//Pausenzeit Rost
		ScalPauseRost.x			:= GesLeistungSoll;
		ScalPauseRost.x1		:= GesLeistungMin;
		ScalPauseRost.x2		:= GesLeistungMax;
		ScalPauseRost.y1		:= RostPauseMin;
		ScalPauseRost.y2		:= RostPauseMax;
		ScalPauseRost();

		//Ausgabe skalierter Sollwert
		SaugzugDrehzSoll		:= ScalDrehzSaugzug.y;
		PrimaerStellSoll		:= ScalStellPrimaer.y;
		SekundaerStellSoll		:= ScalStellSekundaer.y;
		ReziStellSoll			:= ScalStellRezi.y;
		EinschubPulsSoll		:= REAL_TO_UDINT(ScalPulsEinschub.y);
		EinschubPauseSoll		:= REAL_TO_UDINT(ScalPauseEinschub.y);
		RostPulsSoll			:= REAL_TO_UDINT(ScalPulsRost.y);
		RostPauseSoll			:= REAL_TO_UDINT(ScalPauseRost.y);

	ELSE

		SaugzugDrehzSoll		:= 0.0;
		PrimaerStellSoll		:= 0.0;
		SekundaerStellSoll		:= 0.0;
		ReziStellSoll			:= 0.0;
		EinschubPulsSoll		:= 0;
		EinschubPauseSoll		:= 0;
		RostPulsSoll			:= 0;
		RostPauseSoll			:= 0;

	END_IF

END_FUNCTION_BLOCK
```

#### fbLascoZund.st - Funktionsblock Zündgebläse
```iecst
(********************************************************************
 * COPYRIGHT -- LASCO Heu- und Forsttechnik GmbH
 ********************************************************************
 * Library: LascoUtil
 * Datei: fbLascoZund.st
 * Autor: Rudolf Lachner
 * Erstellt: 28. März 2013
 ********************************************************************
 * Implementierung der Library LascoUtil
 ********************************************************************)

(* Funktionsblock Zündgebläse *)
FUNCTION_BLOCK fbLascoZund

	//Max. Zündzeit Zählen
	TON_Zuendzeit(IN := Freigabe, Zeit := Zuendzeit, Tick := Tick);

	IF (Freigabe = TRUE) THEN

		//Zündtemperatur erreicht
		IF (IstTemp > SollTemp) THEN
			Zuendspule 		:= FALSE;
			ZuendungOK 		:= TRUE;
			ZuendungFehler 	:= FALSE;

		//Zündzeit abgelaufen und Temperatur nicht erreicht
		ELSIF (IstTemp < SollTemp AND TON_Zuendzeit.Q) THEN
			Zuendspule 		:= FALSE;
			ZuendungOK 		:= FALSE;
			ZuendungFehler 	:= TRUE;

		//Zündung EIN
		ELSE
			Zuendspule 		:= TRUE;
			ZuendungOK 		:= FALSE;
			ZuendungFehler 	:= FALSE;
		END_IF

		//Nachlaufzeit Zündgebläse
		TOF_Nachlaufzeit(IN := Zuendspule , Zeit := Nachlaufzeit, Tick := Tick);

		Zuendgeblaese := TOF_Nachlaufzeit.Q;

	//Keine Freigabe
	ELSE

		IF (Zuendspule = TRUE) THEN
			Zuendspule := FALSE;
		END_IF

		ZuendungOK 		:= FALSE;
		ZuendungFehler 	:= FALSE;

		//Gebläse läuft auch ohne Freigabe nach
		TOF_Nachlaufzeit(IN := Zuendspule , Zeit := Nachlaufzeit, Tick := Tick);
		Zuendgeblaese := TOF_Nachlaufzeit.Q;

	END_IF

END_FUNCTION_BLOCK
```

#### fbLascoFU.st - Ansteuerung Frequenzumrichter
```iecst
(********************************************************************
 * COPYRIGHT -- LASCO Heu- und Forsttechnik GmbH
 ********************************************************************
 * Library: LascoUtil
 * Datei: fbLascoFU.st
 * Autor: Rudolf Lachner
 * Erstellt: 28. März 2013
 ********************************************************************
 * Implementierung der Library LascoUtil
 ********************************************************************)

(* Ansteuerung Frequenzumrichter *)
FUNCTION_BLOCK fbLascoFU

	//Betriebsmeldung abwarten
	TON_Betriebsmeldung(IN := (Freigabe AND NOT BetrMldg AND NOT Reset AND (SollDrehzahl > 0)), Zeit := AnsprechZeitFU, Tick := Tick);

	//Erster Aufruf
	IF (NOT InitDone) OR Reset THEN
		ResetDone	:= TRUE;
		InitDone	:= TRUE;
	END_IF

	//Keine Betriebsmeldung
	IF (TON_Betriebsmeldung.Q) THEN
		StoerungFU 	:= TRUE;
	END_IF

	//Umrichter Betrieb
	IF (Freigabe AND ResetDone) THEN

		BetriebFU := DrehzahlFU <> 0;

		//Zeit in Millisekunden umrechnen
		RampDownMillis 	:= REAL_TO_DINT(RampeDownSek * 1000);
		RampUpMillis 	:= REAL_TO_DINT(RampeUpSek * 1000);

		//Rampenfunktion
		LCRRamp_0.enable  := Freigabe;
		LCRRamp_0.y_max   := MaxDrehzahl;
		LCRRamp_0.y_min   := MinDrehzahl;
		LCRRamp_0.y_set   := IstDrehzahl;
		LCRRamp_0.set     := EDGEPOS(Init);
		LCRRamp_0.x		  := SollDrehzahl;

		IF (RampUpMillis > 0) THEN
			LCRRamp_0.dy_up   := (MaxDrehzahl - MinDrehzahl)*1000/DINT_TO_REAL(RampUpMillis);
		ELSE
			LCRRamp_0.dy_up   := 999999999;
		END_IF

		IF (RampDownMillis > 0) THEN
			LCRRamp_0.dy_down := (MaxDrehzahl - MinDrehzahl)*1000/DINT_TO_REAL(RampDownMillis);
		ELSE
			LCRRamp_0.dy_down  := 999999999;
		END_IF

		LCRRamp_0();

		IF (LCRRamp_0.dy_down = 999999999 OR LCRRamp_0.dy_up = 999999999) THEN
			DrehzahlFU := SollDrehzahl;
		ELSE
			DrehzahlFU :=	LCRRamp_0.y;
		END_IF

	ELSE

		LCRRamp_0.x		  	:= 0;
		LCRRamp_0.dy_down  	:= 999999999;
		LCRRamp_0();

		BetriebFU 			:= FALSE;
		DrehzahlFU 			:= 0;
	END_IF

	//Störung Reset
	IF (EDGENEG(Freigabe) OR (NOT Freigabe AND NOT BetrMldg) OR Reset OR BetrMldg) THEN
		ResetDone 	:= TRUE;
		StoerungFU 	:= FALSE;
	END_IF

END_FUNCTION_BLOCK
```

#### fbLascoZweiPunktAchse.st - Ansteuerung Zweipunktachse
```iecst
(********************************************************************
 * COPYRIGHT -- LASCO Heu- und Forsttechnik GmbH
 ********************************************************************
 * Library: LascoUtil
 * Datei: fbLascoZweiPunktAchse.st
 * Autor: Rudolf Lachner
 * Erstellt: 28. März 2013
 ********************************************************************
 * Implementierung der Library LascoUtil
 ********************************************************************)

(* Ansteuerung Zweipunktachse *)
FUNCTION_BLOCK fbLascoZweiPunktAchse

	IF (Freigabe AND NOT Stoerung) THEN

		//Minimale Ansprechzeit Anforderung Bewegung Vorwärts
		TON_Ansprechzeit(IN := Vor, Zeit := AnsprechZeit, Tick := Tick);

		//Minimale Laufzeit Aktor Vorwärts
		TOF_Laufzeit(IN := TON_Ansprechzeit.Q, Zeit := MinLaufZeit, Tick := Tick);

		loc_Vor := TOF_Laufzeit.Q;

		//Minimale Ansprechzeit Anforderung Bewegung Rückwärts
		TON_AnsprechzeitZurueck(IN := Zurueck, Zeit := AnsprechZeit, Tick := Tick);

		//Minimale Laufzeit Aktor Rückwärts
		TOF_LaufzeitZurueck(IN := TON_AnsprechzeitZurueck.Q, Zeit := MinLaufZeit, Tick := Tick);

		loc_Zurueck := TOF_LaufzeitZurueck.Q;

		//Vorwärtsbewegung
		IF (loc_Vor AND NOT ESVor AND NOT Stoerung AND NOT loc_Zurueck) THEN
			Motor_Vor 		:= TRUE;
			Motor_Zurueck 	:= FALSE;

		//Rückwärtsbewegung
		ELSIF (loc_Zurueck AND NOT ESZurueck AND NOT Stoerung AND NOT loc_Vor) THEN
			Motor_Vor 		:= FALSE;
			Motor_Zurueck 	:= TRUE;

		//Stillstand
		ELSIF (loc_Zurueck AND NOT ESVor AND NOT Stoerung AND NOT loc_Zurueck) THEN
			Motor_Vor		:= FALSE;
			Motor_Zurueck	:= FALSE;
			loc_Vor			:= FALSE;
			loc_Zurueck		:= FALSE;

		//Stillstand
		ELSE
			Motor_Vor 		:= FALSE;
			Motor_Zurueck 	:= FALSE;
		END_IF

		//Verriegelung
		IF (loc_Vor AND loc_Zurueck) THEN
			Motor_Vor 		:= FALSE;
			Motor_Zurueck 	:= FALSE;
		END_IF

	//Keine Freigabe oder Fehler
	ELSE
		Motor_Vor 		:= FALSE;
		Motor_Zurueck 	:= FALSE;

	END_IF

	//Fehler
	IF ((ESVor AND ESZurueck) OR (Stoerung)) THEN
		Motor_Vor 		:= FALSE;
		Motor_Zurueck 	:= FALSE;
		Fehler 			:= TRUE;

	ELSE
		Fehler 			:= FALSE;
	END_IF

END_FUNCTION_BLOCK
```

#### fbLascoStellachse.st - Ansteuerung Stellachsen
```iecst
(********************************************************************
 * COPYRIGHT -- LASCO Heu- und Forsttechnik GmbH
 ********************************************************************
 * Library: LascoUtil
 * Datei: fbLascoStellachse.st
 * Autor: Rudolf Lachner
 * Erstellt: 29. März 2013
 ********************************************************************
 * Implementierung der Library LascoUtil
 ********************************************************************)

(* Ansteuerung Stellachsen *)
FUNCTION_BLOCK fbLascoStellachse

	IF (Freigabe AND NOT Stoerung) THEN

		//Stellachse zu fahren
		IF (SollStellung < IstStellung - Hysterese AND NOT EsVor) THEN
			MotorVor 		:= FALSE;
			MotorZurueck 	:= TRUE;

		//Stellsachse auf fahren
		ELSIF (SollStellung > IstStellung + Hysterese AND NOT EsZurueck) THEN
			MotorVor 		:= TRUE;
			MotorZurueck 	:= FALSE;

		//Stellachse Aus
		ELSE
			MotorVor 		:= FALSE;
			MotorZurueck 	:= FALSE;
		END_IF
	ELSE
		MotorVor 			:= FALSE;
		MotorZurueck 		:= FALSE;
	END_IF

	//Fehler
	IF ((EsVor AND EsZurueck) OR Stoerung) THEN
		MotorVor 		:= FALSE;
		MotorZurueck 	:= FALSE;
		Fehler 			:= TRUE;
	ELSE
		Fehler 			:= FALSE;
	END_IF

END_FUNCTION_BLOCK
```

#### fbLascoStellachseAnalog.st - Ansteuerung von analogen Stellachsen
```iecst
(********************************************************************
 * COPYRIGHT -- LASCO Heu- und Forsttechnik GmbH
 ********************************************************************
 * Library: LascoUtil
 * Datei: fbStellachseAnalog.st
 * Autor: Rudolf Lachner
 * Erstellt: 29. März 2013
 ********************************************************************
 * Implementierung der Library LascoUtil
 ********************************************************************)

(* Ansteuerung von analogen Stellachsen *)
FUNCTION_BLOCK fbLascoStellachseAnalog

	IF (Freigabe AND NOT Stoerung) THEN

		//Achse verfahren
		IF (SollStellung < IstStellung - Hysterese AND NOT EsVor) THEN
			MotorStellung := SollStellung;
		ELSIF (SollStellung > IstStellung + Hysterese AND NOT EsZurueck) THEN
			MotorStellung := SollStellung;

		//Achse Stillstand
		ELSE
			MotorStellung 	:= IstStellung;
		END_IF
	ELSE
		MotorStellung 		:= IstStellung;
	END_IF

	//Fehler
	IF ((EsVor AND EsZurueck) OR Stoerung) THEN
		MotorStellung 	:= IstStellung;
		Fehler 			:= TRUE;
	ELSE
		Fehler 			:= FALSE;
	END_IF

END_FUNCTION_BLOCK
```

#### fbLascoStellachseDigital.st - Ansteuerung von Stellachsen ohne Positionsrückmeldung
```iecst
(********************************************************************
 * COPYRIGHT -- LASCO Heu- und Forsttechnik GmbH
 ********************************************************************
 * Library: LascoUtil
 * Datei: fbLascoStellachseDigital.st
 * Autor: Rudolf Lachner
 * Erstellt: 7. Januar 2014
 ********************************************************************
 * Implementierung der Library LascoUtil
 ********************************************************************)

(* Ansteuerung von Stellachsen ohne Positionsrückmeldung *)
FUNCTION_BLOCK fbLascoStellachseDigital

	//Eingänge
	LCRContinServo_0.enable			:= Freigabe;
	LCRContinServo_0.ref			:= Referenz;
	LCRContinServo_0.min_value		:= MinPosition;
	LCRContinServo_0.max_value		:= MaxPosition;
	LCRContinServo_0.t_change_up	:= Oeffnungszeit;
	LCRContinServo_0.t_change_down	:= Schliesszeit;
	LCRContinServo_0.t_impulse		:= MinImpulsdauer;
	LCRContinServo_0.x				:= Sollstellung;
	LCRContinServo_0();

	//Ausgänge
	MotorAuf		:= LCRContinServo_0.up;
	MotorZu			:= LCRContinServo_0.down;
	ReferenzAktiv	:= Referenz AND NOT ReferenzOk;

	IF (EDGEPOS(LCRContinServo_0.refOk)) THEN
		ReferenzOk		:= TRUE;
	ELSIF (NOT Freigabe) THEN
		ReferenzOk		:= FALSE;
	END_IF

	//Weg pro Sekunde/10 errechnen
	//****************************
	IF (Oeffnungszeit <> 0) THEN
		WegProZeitAuf	:= ((MaxPosition - MinPosition) / Oeffnungszeit) / 10;
	END_IF
	IF (Schliesszeit <> 0) THEN
		WegProZeitZu	:= ((MaxPosition - MinPosition) / Schliesszeit) / 10;
	END_IF

	//Ist- Position Klappe errechnen
	IF (ReferenzAktiv) THEN
		IstPosition		:= MinPosition;
	ELSIF (EDGEPOS(ReferenzOk)) THEN
		IstPosition		:= MinPosition;
	ELSIF (IstPosition < MinPosition) THEN
		IstPosition		:= MinPosition;
	ELSIF (IstPosition > MaxPosition) THEN
		IstPosition		:= MaxPosition;
	ELSIF (MotorAuf AND Tick AND ReferenzOk AND (IstPosition < MaxPosition)) THEN
		IstPosition		:= IstPosition + WegProZeitAuf;
	ELSIF (MotorZu AND Tick AND ReferenzOk AND (IstPosition > MinPosition)) THEN
		IstPosition		:= IstPosition - WegProZeitZu;
	END_IF

END_FUNCTION_BLOCK
```

#### fbLascoWarmluftsteller.st - Ansteuerung Warmluftgebläse mit Kühlreduzierung
```iecst
(********************************************************************
 * COPYRIGHT -- LASCO Heu- und Forsttechnik GmbH
 ********************************************************************
 * Library: LascoUtil
 * Datei: fbLascoWarmluftsteller.st
 * Autor: Rudolf Lachner
 * Erstellt: 29. März 2013
 ********************************************************************
 * Implementierung der Library LascoUtil
 ********************************************************************)

(* Ansteuerung Warmluftgebläse mit Kühlreduzierung *)
FUNCTION_BLOCK fbLascoWarmluftsteller

	IF (Freigabe) THEN

		//Schrittschaltwerk Kühlreduzierung
		//=================================

		curState	:= nextState;

		CASE curState OF

			//****************************************************************************************************************************************************************************
			0://NORMAL

				//*** state entry ***
				IF (stateEntry = TRUE) THEN
					stateEntry := FALSE;
				END_IF

				//*** state during ***
				locDrehzahl1 	:= WLG1SollDRZ;
				locDrehzahl2 	:= WLG2SollDRZ;
				WLG1DRZStell 	:= locDrehzahl1;
				WLG2DRZStell  	:= locDrehzahl2;

				//*** state exit ***
				IF (IstTemperatur < GrenzTemperatur) THEN
					nextState 	:= 1;
					stateEntry 	:= TRUE;
				ELSE
					nextState := curState;
				END_IF

			//********************************************************************************************************************************************************************************************
			1://DREHZAHL MINDERUNG

				//*** state entry ***
				IF (stateEntry = TRUE) THEN
					stateEntry := FALSE;
					IF (((locDrehzahl1 - MinderungDRZ) > WLG1MinDRZ) AND ((locDrehzahl2 - MinderungDRZ) > WLG2MinDRZ)) THEN
						locDrehzahl1 := locDrehzahl1 - MinderungDRZ;
						locDrehzahl2 := locDrehzahl2 - MinderungDRZ;
					ELSE
						locDrehzahl1 := WLG1MinDRZ;
						locDrehzahl2 := WLG2MinDRZ;
					END_IF
					TON_WarmluftSteller.IN		:= TRUE;
					TON_WarmluftSteller.Zeit	:= Bezugszeit;
				END_IF

				//*** state during ***

				//Zeit starten
				TON_WarmluftSteller.Tick	:= Tick;

				IF ((WLG1SollDRZ < locDrehzahl1) AND (WLG2SollDRZ < locDrehzahl2)) THEN
					locDrehzahl1 := WLG1SollDRZ;
					locDrehzahl2 := WLG2SollDRZ;
				END_IF

				WLG1DRZStell := locDrehzahl1;
				WLG2DRZStell := locDrehzahl2;

				//*** state exit ***

				//Bezugszeit abgelaufen, weiter reduzieren
				IF ((TON_WarmluftSteller.Q) AND (IstTemperatur <= GrenzTemperatur)) THEN
					nextState 				:= 1;
					stateEntry 				:= TRUE;
					TON_WarmluftSteller.IN 	:= FALSE;

					//Bezugszeit abgelaufen, wieder erhöhen
				ELSIF ((TON_WarmluftSteller.Q) AND (IstTemperatur > GrenzTemperatur)) THEN
					nextState 				:= 2;
					stateEntry 				:= TRUE;
					TON_WarmluftSteller.IN 	:= FALSE;
				ELSE
					nextState := curState;
				END_IF

			//****************************************************************************************************************************************************************************************************************
			2://DREHZAHL ERHÖHEN

				//*** state entry ***
				IF (stateEntry = TRUE) THEN
					stateEntry := FALSE;
					IF ((locDrehzahl1 < WLG1MinDRZ) AND (locDrehzahl2 < WLG2MinDRZ))THEN
						locDrehzahl1 := WLG1MinDRZ;
						locDrehzahl2 := WLG2MinDRZ;
					END_IF
					IF (((locDrehzahl1 + MinderungDRZ) < WLG1SollDRZ) AND
						((locDrehzahl2 + MinderungDRZ) < WLG2SollDRZ)) THEN
						locDrehzahl1 := locDrehzahl1 + MinderungDRZ;
						locDrehzahl2 := locDrehzahl2 + MinderungDRZ;
					ELSE
						locDrehzahl1 := WLG1SollDRZ;
						locDrehzahl2 := WLG2SollDRZ;
					END_IF
					TON_WarmluftSteller.IN 		:= TRUE;
					TON_WarmluftSteller.Zeit 	:= Bezugszeit;
				END_IF

				//*** state during ***
				TON_WarmluftSteller.Tick	:= Tick;
				WLG1DRZStell				:= locDrehzahl1;
				WLG2DRZStell				:= locDrehzahl2;

				//*** state exit ***
				IF ((locDrehzahl1 >= WLG1SollDRZ) AND (locDrehzahl2 >= WLG2SollDRZ)) THEN
					nextState 				:= 0;
					stateEntry 				:= TRUE;
					TON_WarmluftSteller.IN 	:= FALSE;

				ELSIF ((TON_WarmluftSteller.Q = TRUE) AND (IstTemperatur <= GrenzTemperatur)) THEN
					nextState 				:= 1;
					stateEntry 				:= TRUE;
					TON_WarmluftSteller.IN 	:= FALSE;

				ELSIF ((TON_WarmluftSteller.Q = TRUE) AND (IstTemperatur > GrenzTemperatur)) THEN
					nextState 				:= 2;
					stateEntry 				:= TRUE;
					TON_WarmluftSteller.IN 	:= FALSE;

				ELSE
					nextState := curState;
				END_IF

		END_CASE

	ELSE

		nextState 				:= 0;
		locDrehzahl1 			:= 0.0;
		locDrehzahl2 			:= 0.0;
		WLG1DRZStell 			:= 0.0;
		WLG2DRZStell 			:= 0.0;
		TON_WarmluftSteller.IN 	:= FALSE;

	END_IF

	TON_WarmluftSteller();

END_FUNCTION_BLOCK
```

#### fbLascoFreilauf.st - Freilauffunktion für blockierende Motoren
```iecst
(********************************************************************
 * COPYRIGHT -- LASCO Heu- und Forsttechnik GmbH
 ********************************************************************
 * Library: LascoUtil
 * Datei: fbLascoFreilauf.st
 * Autor: Rudolf Lachner
 * Erstellt: 30. März 2013
 ********************************************************************
 * Implementierung der Library LascoUtil
 ********************************************************************)

(* Freilauffunktion für blockierende Motoren *)
FUNCTION_BLOCK fbLascoFreilauf

	IF (Freigabe) THEN

		//Drehbewegung überwachen
		DRZWaechter.Motor	:= MotorVor;
		DRZWaechter.Impuls	:= Impuls;
		DRZWaechter.Tick	:= Tick;
		DRZWaechter.Zeit	:= Stehzeit;
		DRZWaechter.Quit	:= NOT MotorVor;

		curStep		:= nextStep;

		//Schrittschaltwerk Freilauffunktion
		//==================================

		CASE curStep OF

			//******************************************************************************************************************************************************************
			0://NORMAL

				//*** state entry ***
				IF (stateEntry = TRUE) THEN
					CounterVersuche		:= CounterVersuche + 1;
					stateEntry			:= FALSE;
					TON_ResetCounter.IN	:= TRUE;
				END_IF

				//*** state during ***
				MotorVor		:= TRUE;
				MotorZurueck	:= FALSE;

				//Zähler rücksetzen
				IF (TON_ResetCounter.Q = TRUE) THEN
					CounterVersuche	:= 0;
				END_IF

				//*** state exit ***
				IF (DRZWaechter.Fehler = TRUE) AND (CounterVersuche < MaxVersuche) THEN
					stateEntry			:= TRUE;
					TON_ResetCounter.IN	:= FALSE;
					nextStep			:= 1;
				ELSIF (DRZWaechter.Fehler = TRUE) THEN
					stateEntry			:= TRUE;
					TON_ResetCounter.IN	:= FALSE;
					nextStep			:= 4;
				ELSE
					nextStep	:= curStep;
				END_IF

			//******************************************************************************************************************************************************************************
			1://VERZÖGERUNG FREILAUF

				//*** state entry ***
				IF (stateEntry = TRUE) THEN
					stateEntry		:= FALSE;
					TON_VerzRW.IN	:= TRUE;
				END_IF

				//*** state during ***
				MotorVor		:= FALSE;
				MotorZurueck	:= FALSE;

				//... Verzögerung abwarten

				//*** state exit ***
				IF (TON_VerzRW.Q = TRUE) THEN
					stateEntry		:= TRUE;
					TON_VerzRW.IN	:= FALSE;
					nextStep		:= 2;
				ELSE
					nextStep		:= curStep;
				END_IF

			//**********************************************************************************************************************************************************************************
			2://FREILAUF

				//*** state entry ***
				IF (stateEntry = TRUE) THEN
					stateEntry			:= FALSE;
					TON_Freilaufzeit.IN	:= TRUE;
				END_IF

				//*** state during ***
				MotorVor		:= FALSE;
				MotorZurueck	:= TRUE;

				//... Freilaufzeit abwarten

				//*** state exit ***
				IF (TON_Freilaufzeit.Q	= TRUE) THEN
					stateEntry			:= TRUE;
					TON_Freilaufzeit.IN	:= FALSE;
					nextStep			:= 3;
				ELSE
					nextStep			:= curStep;
				END_IF

			//********************************************************************************************************************************************************************************************
			3://VERZÖGERUNG NACH FREILAUF

				//*** state entry ***
				IF (stateEntry = TRUE) THEN
					stateEntry		:= FALSE;
					TON_VerzRW.IN	:= TRUE;
				END_IF

				//*** state during ***
				MotorVor		:= FALSE;
				MotorZurueck	:= FALSE;

				//... Verzögerung abwarten

				//*** state exit ***
				IF (TON_VerzRW.Q = TRUE) THEN
					stateEntry		:= TRUE;
					TON_VerzRW.IN	:= FALSE;
					nextStep		:= 0;
				ELSE
					nextStep		:= curStep;
				END_IF

			//***********************************************************************************************************************************************************************************************
			4://FEHLER

				//*** state entry ***
				IF (stateEntry = TRUE) THEN
					Fehler			:= TRUE;
					CounterVersuche	:= 0;
					stateEntry		:= FALSE;
				END_IF

				//*** state during ***
				MotorVor		:= FALSE;
				MotorZurueck	:= FALSE;

				//... Quittierung abwarten

				//*** state exit ***
				IF (Quit = TRUE) THEN
					Fehler		:= FALSE;
					nextStep	:= 0;
				ELSE
					nextStep	:= curStep;
				END_IF

		END_CASE

	//Keine Freigabe
	ELSE

		MotorVor			:= FALSE;
		MotorZurueck		:= FALSE;
		TON_VerzRW.IN		:= FALSE;
		TON_Freilaufzeit.IN	:= FALSE;
		TON_ResetCounter.IN	:= FALSE;
		CounterVersuche		:= 0;
		Fehler				:= FALSE;
		nextStep			:= 0;
		curStep				:= 0;
	END_IF

		//Funtionsblöcke aufrufen
		//=======================

		//Drehzahlüberwachung
		DRZWaechter();

		//TON Verzögerung Richtungswechsel
		TON_VerzRW.Tick	:= Tick;
		TON_VerzRW.Zeit	:= VerzFreilauf;
		TON_VerzRW();

		//TON Freilaufzeit
		TON_Freilaufzeit.Tick	:= Tick;
		TON_Freilaufzeit.Zeit	:= Freilaufzeit;
		TON_Freilaufzeit();

		//TON Quittierung Zähler
		TON_ResetCounter.Tick	:= Tick;
		TON_ResetCounter.Zeit	:= 60.0;
		TON_ResetCounter();

END_FUNCTION_BLOCK
```

#### fbLascoBrStfLst.st - Berechnung der Brennstoffleistung
```iecst
(********************************************************************
 * COPYRIGHT -- LASCO Heu- und Forsttechnik GmbH
 ********************************************************************
 * Library: LascoUtil
 * Datei: fbLascoBrStfLst.st
 * Autor: Rudolf Lachner
 * Erstellt: 11. Dezember 2013
 ********************************************************************
 * Implementierung der Library LascoUtil
 ********************************************************************)

(* Berechnung der Brennstoffleistung *)
FUNCTION_BLOCK fbLascoBrStfLst

	IF (sekTick) THEN

		LeistungSek		:= LeistungAkt / 3600;
		Leistung_kWh	:= Leistung_kWh + LeistungSek;

		IF (Leistung_kWh >= 10) THEN
			Leistung_kWh	:= Leistung_kWh - 10;
			Leistung_MWh	:= Leistung_MWh + 1;
		END_IF
	END_IF

	IF (Reset) THEN
		Leistung_kWh	:= 0;
		Leistung_MWh	:= 0;
	END_IF

END_FUNCTION_BLOCK
```

#### fbLascoFuellst.st - Überwachung von Fuellstandssensoren
```iecst
(********************************************************************
 * COPYRIGHT -- LASCO Heu- und Forsttechnik GmbH
 ********************************************************************
 * Library: LascoUtil
 * Datei: fbLascoFuellst.st
 * Autor: Rudolf Lachner
 * Erstellt: 13. Januar 2014
 ********************************************************************
 * Implementierung der Library LascoUtil
 ********************************************************************)

(* Überwachung von Fuellstandssensoren *)
FUNCTION_BLOCK fbLascoFuellst

	IF (EDGE(Fuellstand)) THEN
		cKeineFlankeFs	:= 0;
	ELSIF (EinschubEin) AND (NOT Fehler) THEN
		cKeineFlankeFs	:= cKeineFlankeFs + Tick;
	END_IF

	IF (Quit) THEN
		Fehler			:= FALSE;
		cKeineFlankeFs	:= 0;
	ELSIF (cKeineFlankeFs >= VerzZeit) AND (VerzZeit > 0) THEN
		Fehler			:= TRUE;
	END_IF

END_FUNCTION_BLOCK
```

#### fbLascoWlg.st - Ansteuerung für Warmluftgebläse ohne Drehzahlvorgabe
```iecst
(********************************************************************
 * COPYRIGHT -- LASCO Heu- und Forsttechnik GmbH
 ********************************************************************
 * Library: LascoUtil
 * Datei: fbLascoWlg.st
 * Autor: Rudolf Lachner
 * Erstellt: 15. Januar 2014
 ********************************************************************
 * Implementierung der Library LascoUtil
 ********************************************************************)

(* Ansteuerung für Warmluftgebläse ohne Drehzahlvorgabe *)
FUNCTION_BLOCK fbLascoWlg

	IF (Freigabe AND NOT Stoerung) THEN

		//Temperatur unter Min -> Stopp
		IF (IstTemp <= StopBeiTemp) THEN
			GeblaeseEin	:= FALSE;
			//Temperatur über Max -> Start
		ELSIF (IstTemp >= StartBeiTemp) AND (StartBeiTemp <> 0) THEN
			GeblaeseEin	:= TRUE;
		END_IF

	ELSE

		GeblaeseEin	:= FALSE;

	END_IF

	IF (Stoerung) THEN
		Fehler		:= TRUE;
	ELSE
		Fehler		:= FALSE;
	END_IF

END_FUNCTION_BLOCK
```

#### fbLascoBmin.st - Betriebsdauer in Minuten zählen
```iecst
(********************************************************************
 * COPYRIGHT -- LASCO Heu- und Forsttechnik GmbH
 ********************************************************************
 * Library: LascoUtil
 * Datei: fbLascoBmin.st
 * Autor: Rudolf Lachner
 * Erstellt: 16. Januar 2014
 ********************************************************************
 * Implementierung der Library LascoUtil
 ********************************************************************)

(* Betriebsdauer in Minuten zählen *)
FUNCTION_BLOCK fbLascoBmin

	IF (Aktiv AND sekTick) THEN
		IF (Sekunden < 59) THEN
			Sekunden	:= Sekunden + 1;
		ELSE
			Minuten		:= Minuten + 1;
			Sekunden	:= 0;
		END_IF
	END_IF

	IF (Reset) THEN
		Sekunden	:= 0;
		Minuten		:= 0;
	END_IF

END_FUNCTION_BLOCK
```

#### fbLascoStdMin.st - Angehängte Betriebsdauer von Minuten in Stunden umwandeln
```iecst
(********************************************************************
 * COPYRIGHT -- LASCO Heu- und Forsttechnik GmbH
 ********************************************************************
 * Library: LascoUtil
 * Datei: fbLascoStdMin.st
 * Autor: Rudolf Lachner
 * Erstellt: 16. Januar 2014
 ********************************************************************
 * Implementierung der Library LascoUtil
 ********************************************************************)

(* Angehängte Betriebsdauer von Minuten in Stunden umwandeln *)
FUNCTION_BLOCK fbLascoStdMin

	IF (Minuten > 59) THEN
		Stunden		:= Stunden + 1;
		Minuten		:= 0;
	END_IF

	IF (Reset) THEN
		Stunden		:= 0;
		Minuten		:= 0;
	END_IF

END_FUNCTION_BLOCK
```
